  MoveL 1972 to (37.53, 7.97, 0.25) mm, rotated rx 180 ry 0 rz 90 deg; joints [74.413, -17.204, 82.136, 0, 25.068, 74.413]
  MoveL 1973 to (38.64, 6.94, -0.16) mm, rotated rx 180 ry 0 rz 90 deg; joints [74.39, -17.155, 82.02, 0, 25.135, 74.39]
  MoveL 1974 to (39.97, 6.21, -0.56) mm, rotated rx 180 ry 0 rz 90 deg; joints [74.379, -17.103, 81.894, 0, 25.209, 74.379]
  MoveL 1975 to (41.44, 5.79, -0.97) mm, rotated rx -180 ry 0 rz 90 deg; joints [74.379, -17.051, 81.765, 0, 25.286, 74.379]
  MoveL 1976 to (42.95, 5.71, -1.37) mm, rotated rx 180 ry 0 rz 90 deg; joints [74.389, -16.999, 81.638, 0, 25.361, 74.389]
  MoveL 1977 to (44.45, 5.96, -1.78) mm, rotated rx 180 ry 0 rz 90 deg; joints [74.411, -16.949, 81.519, 0, 25.43, 74.411]
  MoveL 1978 to (45.85, 6.54, -2.19) mm, rotated rx 180 ry 0 rz 90 deg; joints [74.441, -16.903, 81.414, 0, 25.489, 74.441]
  MoveL 1979 to (47.1, 7.42, -2.59) mm, rotated rx 180 ry 0 rz 90 deg; joints [74.48, -16.862, 81.327, 0, 25.535, 74.48]
  MoveL 1980 to (48.09, 8.56, -3) mm, rotated rx 180 ry 0 rz 90 deg; joints [74.525, -16.827, 81.263, 0, 25.564, 74.525]
  MoveL 1981 to (59.23, 24.09, -3) mm, rotated rx 180 ry 0 rz 90 deg; joints [75.111, -16.683, 80.75, 0, 25.933, 75.111]
  MoveL 1982 to (60.04, 25.3, -3) mm, rotated rx 180 ry 0 rz 90 deg; joints [75.156, -16.673, 80.714, 0, 25.959, 75.156]
  MoveC 1983 to (60.83, 30.5, -3) mm, rotated rx 180 ry 0 rz 90 deg; joints [75.327, -16.685, 80.757, 0, 25.928, 75.327] to (57.33, 34.43, -3) mm, rotated rx 180 ry 0 rz 90 deg; joints [75.423, -16.78, 81.093, 0, 25.686, 75.423]
  MoveC 1984 to (55.77, 34.77, -3) mm, rotated rx -180 ry 0 rz 90 deg; joints [75.421, -16.814, 81.216, 0, 25.598, 75.421] to (54.17, 34.86, -3) mm, rotated rx -180 ry 0 rz 90 deg; joints [75.41, -16.848, 81.336, 0, 25.512, 75.41]
  MoveL 1985 to (7.66, 33.6, -3) mm, rotated rx 180 ry 0 rz 90 deg; joints [74.974, -17.751, 84.687, 0, 23.065, 74.974]
  MoveC 1986 to (4.92, 33.05, -3) mm, rotated rx -180 ry 0 rz 90 deg; joints [74.933, -17.799, 84.871, 0, 22.928, 74.933] to (2.52, 31.63, -3) mm, rotated rx -180 ry 0 rz 90 deg; joints [74.865, -17.836, 85.014, 0, 22.822, 74.865]
  MoveC 1987 to (0.88, 28.58, -3) mm, rotated rx 180 ry 0 rz 90 deg; joints [74.751, -17.851, 85.072, 0, 22.779, 74.751] to (1.07, 25.11, -3) mm, rotated rx -180 ry 0 rz 90 deg; joints [74.64, -17.83, 84.991, 0, 22.839, 74.64]
  MoveL 1988 to (1.71, 23.22, -3) mm, rotated rx 180 ry 0 rz 90 deg; joints [74.584, -17.809, 84.909, 0, 22.9, 74.584]
  MoveL 1989 to (7.22, 8.05, -3) mm, rotated rx -180 ry 0 rz 90 deg; joints [74.142, -17.629, 84.216, 0, 23.413, 74.142]
  MoveL 1990 to (7.43, 7.5, -3) mm, rotated rx -180 ry 0 rz 90 deg; joints [74.126, -17.622, 84.189, 0, 23.432, 74.126]
  MoveC 1991 to (8.35, 5.81, -3) mm, rotated rx 180 ry 0 rz 90 deg; joints [74.08, -17.595, 84.09, 0, 23.506, 74.08] to (9.69, 4.43, -3) mm, rotated rx -180 ry 0 rz 90 deg; joints [74.048, -17.563, 83.966, 0, 23.597, 74.048]
  MoveL 1992 to (26.06, -8.32, -3) mm, rotated rx 180 ry 0 rz 90 deg; joints [73.791, -17.176, 82.524, 0, 24.652, 73.791]
  MoveL 1993 to (27.21, -9.18, -3) mm, rotated rx 180 ry 0 rz 90 deg; joints [73.774, -17.148, 82.422, 0, 24.726, 73.774]
  MoveC 1994 to (31.85, -10.43, -3) mm, rotated rx 180 ry 0 rz 90 deg; joints [73.778, -17.048, 82.058, 0, 24.99, 73.778] to (36.06, -8.1, -3) mm, rotated rx -180 ry 0 rz 90 deg; joints [73.89, -16.977, 81.801, 0, 25.176, 73.89]
  MoveL 1995 to (36.86, -7.11, -3) mm, rotated rx -180 ry 0 rz 90 deg; joints [73.929, -16.966, 81.763, 0, 25.204, 73.929]
  MoveL 1996 to (44.07, 2.95, -3) mm, rotated rx -180 ry 0 rz 90 deg; joints [74.312, -16.878, 81.444, 0, 25.434, 74.312]
  MoveL 1997 to (48.09, 8.56, -3) mm, rotated rx 180 ry 0 rz 90 deg; joints [74.525, -16.827, 81.263, 0, 25.564, 74.525]
  MoveL 1998 to (41.96, 12.96, -3) mm, rotated rx -180 ry 0 rz 90 deg; joints [74.611, -16.978, 81.804, 0, 25.174, 74.611]
  MoveL 1999 to (41.96, 12.96, 0) mm, rotated rx 180 ry 0 rz 90 deg; joints [74.611, -17.13, 81.905, 0, 25.225, 74.611]
  Establecer velocidad (1000.0 mm/s)
  MoveL 2000 to (41.96, 12.96, 10) mm, rotated rx 180 ry 0 rz 90 deg; joints [74.611, -17.635, 82.239, 0, 25.396, 74.611]
  Establecer velocidad (66.7 mm/s)
  MoveL 2001 to (27.12, 70.14, 10) mm, rotated rx -180 ry 0 rz 90 deg; joints [76.326, -18.224, 84.396, 0, 23.829, 76.326]
  MoveL 2002 to (27.12, 70.14, 0.25) mm, rotated rx -180 ry 0 rz 90 deg; joints [76.326, -17.727, 84.071, 0, 23.656, 76.326]
  MoveL 2003 to (27.33, 71.65, -0.16) mm, rotated rx 180 ry 0 rz 90 deg; joints [76.377, -17.71, 84.069, 0, 23.641, 76.377]
  MoveL 2004 to (27.16, 73.16, -0.56) mm, rotated rx -180 ry 0 rz 90 deg; joints [76.425, -17.699, 84.094, 0, 23.606, 76.425]
  MoveL 2005 to (26.67, 74.59, -0.97) mm, rotated rx 180 ry 0 rz 90 deg; joints [76.468, -17.694, 84.14, 0, 23.554, 76.468]
  MoveL 2006 to (25.87, 75.89, -1.37) mm, rotated rx 180 ry 0 rz 90 deg; joints [76.504, -17.695, 84.207, 0, 23.488, 76.504]
  MoveL 2007 to (24.81, 76.97, -1.78) mm, rotated rx -180 ry 0 rz 90 deg; joints [76.531, -17.699, 84.288, 0, 23.411, 76.531]
  MoveL 2008 to (23.53, 77.8, -2.19) mm, rotated rx 180 ry 0 rz 90 deg; joints [76.547, -17.706, 84.381, 0, 23.325, 76.547]
  MoveL 2009 to (22.1, 78.32, -2.59) mm, rotated rx 180 ry 0 rz 90 deg; joints [76.553, -17.715, 84.479, 0, 23.236, 76.553]
  MoveL 2010 to (20.6, 78.48, -3) mm, rotated rx -180 ry 0 rz 90 deg; joints [76.547, -17.723, 84.576, 0, 23.147, 76.547]
  MoveC 2011 to (-4.88, 78.78, -3) mm, rotated rx 180 ry 0 rz 90 deg; joints [76.355, -18.184, 86.391, 0, 21.793, 76.355] to (-30.36, 79, -3) mm, rotated rx -180 ry 0 rz 90 deg; joints [76.153, -18.615, 88.168, 0, 20.446, 76.153]
  MoveC 2012 to (-33.55, 78.8, -3) mm, rotated rx -180 ry 0 rz 90 deg; joints [76.12, -18.665, 88.385, 0, 20.281, 76.12] to (-36.69, 78.18, -3) mm, rotated rx 180 ry 0 rz 90 deg; joints [76.073, -18.713, 88.59, 0, 20.124, 76.073]
  MoveC 2013 to (-40.07, 74.26, -3) mm, rotated rx 180 ry 0 rz 90 deg; joints [75.912, -18.752, 88.754, 0, 19.997, 75.912] to (-39.33, 69.14, -3) mm, rotated rx 180 ry 0 rz 90 deg; joints [75.745, -18.719, 88.615, 0, 20.104, 75.745]
  MoveC 2014 to (-37.7, 67.63, -3) mm, rotated rx 180 ry 0 rz 90 deg; joints [75.709, -18.687, 88.477, 0, 20.21, 75.709] to (-35.91, 66.33, -3) mm, rotated rx 180 ry 0 rz 90 deg; joints [75.68, -18.653, 88.331, 0, 20.322, 75.68]
  MoveL 2015 to (-32.69, 64.28, -3) mm, rotated rx 180 ry 0 rz 90 deg; joints [75.639, -18.592, 88.074, 0, 20.518, 75.639]
  MoveL 2016 to (-16.58, 54.08, -3) mm, rotated rx 180 ry 0 rz 90 deg; joints [75.437, -18.279, 86.776, 0, 21.503, 75.437]
  MoveL 2017 to (-12.87, 51.72, -3) mm, rotated rx -180 ry 0 rz 90 deg; joints [75.391, -18.205, 86.473, 0, 21.731, 75.391]
  MoveC 2018 to (-9.92, 50.46, -3) mm, rotated rx 180 ry 0 rz 90 deg; joints [75.375, -18.148, 86.244, 0, 21.903, 75.375] to (-6.73, 50.2, -3) mm, rotated rx 180 ry 0 rz 90 deg; joints [75.393, -18.09, 86.015, 0, 22.075, 75.393]
  MoveC 2019 to (32.51, 53.09, -3) mm, rotated rx -180 ry 0 rz 90 deg; joints [75.816, -17.376, 83.265, 0, 24.111, 75.816] to (71.77, 55.83, -3) mm, rotated rx 180 ry 0 rz 90 deg; joints [76.217, -16.589, 80.419, 0, 26.17, 76.217]
  MoveC 2020 to (75.27, 57.49, -3) mm, rotated rx -180 ry 0 rz 90 deg; joints [76.296, -16.522, 80.186, 0, 26.336, 76.296] to (76.7, 61.09, -3) mm, rotated rx 180 ry 0 rz 90 deg; joints [76.421, -16.511, 80.145, 0, 26.366, 76.421]
  MoveL 2021 to (76.7, 71.55, -3) mm, rotated rx -180 ry 0 rz 90 deg; joints [76.753, -16.564, 80.332, 0, 26.232, 76.753]
  MoveL 2022 to (76.69, 72.49, -3) mm, rotated rx -180 ry 0 rz 90 deg; joints [76.783, -16.569, 80.35, 0, 26.219, 76.783]
  MoveC 2023 to (75.13, 76.06, -3) mm, rotated rx 180 ry 0 rz 90 deg; joints [76.884, -16.62, 80.53, 0, 26.091, 76.884] to (71.55, 77.57, -3) mm, rotated rx -180 ry 0 rz 90 deg; joints [76.906, -16.704, 80.825, 0, 25.879, 76.906]
  MoveC 2024 to (46.07, 78.07, -3) mm, rotated rx -180 ry 0 rz 90 deg; joints [76.73, -17.23, 82.722, 0, 24.508, 76.73] to (20.6, 78.48, -3) mm, rotated rx -180 ry 0 rz 90 deg; joints [76.547, -17.723, 84.576, 0, 23.147, 76.547]
  MoveL 2025 to (20.49, 70.93, -3) mm, rotated rx 180 ry 0 rz 90 deg; joints [76.299, -17.691, 84.453, 0, 23.238, 76.299]
  MoveL 2026 to (20.49, 70.93, 0) mm, rotated rx 180 ry 0 rz 90 deg; joints [76.299, -17.844, 84.554, 0, 23.29, 76.299]
  Establecer velocidad (1000.0 mm/s)
  MoveL 2027 to (20.49, 70.93, 10) mm, rotated rx -180 ry 0 rz 90 deg; joints [76.299, -18.355, 84.886, 0, 23.468, 76.299]
  Establecer velocidad (66.7 mm/s)
  MoveL 2028 to (27.11, 69.78, 10) mm, rotated rx -180 ry 0 rz 90 deg; joints [76.314, -18.223, 84.39, 0, 23.833, 76.314]
  MoveL 2029 to (27.11, 69.78, 0) mm, rotated rx 180 ry 0 rz 90 deg; joints [76.314, -17.713, 84.057, 0, 23.656, 76.314]
  MoveL 2030 to (27.32, 71.29, -0.41) mm, rotated rx -180 ry 0 rz 90 deg; joints [76.365, -17.696, 84.055, 0, 23.641, 76.365]
  MoveL 2031 to (27.16, 72.8, -0.81) mm, rotated rx -180 ry 0 rz 90 deg; joints [76.413, -17.685, 84.079, 0, 23.606, 76.413]
  MoveL 2032 to (26.67, 74.24, -1.22) mm, rotated rx 180 ry 0 rz 90 deg; joints [76.456, -17.68, 84.126, 0, 23.554, 76.456]
  MoveL 2033 to (25.87, 75.53, -1.63) mm, rotated rx -180 ry 0 rz 90 deg; joints [76.492, -17.68, 84.192, 0, 23.488, 76.492]
  MoveL 2034 to (24.81, 76.62, -2.03) mm, rotated rx 180 ry 0 rz 90 deg; joints [76.519, -17.685, 84.274, 0, 23.411, 76.519]
  MoveL 2035 to (23.53, 77.44, -2.44) mm, rotated rx -180 ry 0 rz 90 deg; joints [76.536, -17.692, 84.367, 0, 23.325, 76.536]
  MoveL 2036 to (22.1, 77.96, -2.84) mm, rotated rx -180 ry 0 rz 90 deg; joints [76.542, -17.7, 84.465, 0, 23.236, 76.542]
  MoveL 2037 to (20.59, 78.12, -3.25) mm, rotated rx 180 ry 0 rz 90 deg; joints [76.535, -17.708, 84.562, 0, 23.147, 76.535]
  MoveC 2038 to (-5.1, 78.43, -3.25) mm, rotated rx -180 ry 0 rz 90 deg; joints [76.341, -18.174, 86.392, 0, 21.782, 76.341] to (-30.8, 78.63, -3.25) mm, rotated rx 180 ry 0 rz 90 deg; joints [76.137, -18.607, 88.184, 0, 20.423, 76.137]
  MoveC 2039 to (-33.67, 78.43, -3.25) mm, rotated rx -180 ry 0 rz 90 deg; joints [76.107, -18.653, 88.378, 0, 20.275, 76.107] to (-36.48, 77.81, -3.25) mm, rotated rx 180 ry 0 rz 90 deg; joints [76.062, -18.695, 88.561, 0, 20.135, 76.062]
  MoveC 2040 to (-39.45, 73.96, -3.25) mm, rotated rx 180 ry 0 rz 90 deg; joints [75.907, -18.727, 88.698, 0, 20.029, 75.907] to (-38.79, 69.14, -3.25) mm, rotated rx 180 ry 0 rz 90 deg; joints [75.75, -18.698, 88.57, 0, 20.128, 75.75]
  MoveC 2041 to (-37.24, 67.74, -3.25) mm, rotated rx 180 ry 0 rz 90 deg; joints [75.716, -18.667, 88.439, 0, 20.228, 75.716] to (-35.54, 66.53, -3.25) mm, rotated rx -180 ry 0 rz 90 deg; joints [75.69, -18.635, 88.301, 0, 20.334, 75.69]
  MoveL 2042 to (-12.65, 52.03, -3.25) mm, rotated rx -180 ry 0 rz 90 deg; joints [75.403, -18.189, 86.455, 0, 21.734, 75.403]
  MoveC 2043 to (-9.84, 50.82, -3.25) mm, rotated rx 180 ry 0 rz 90 deg; joints [75.387, -18.135, 86.236, 0, 21.899, 75.387] to (-6.79, 50.56, -3.25) mm, rotated rx 180 ry 0 rz 90 deg; joints [75.405, -18.08, 86.018, 0, 22.062, 75.405]
  MoveC 2044 to (32.37, 53.44, -3.25) mm, rotated rx -180 ry 0 rz 90 deg; joints [75.827, -17.368, 83.274, 0, 24.094, 75.827] to (71.55, 56.18, -3.25) mm, rotated rx -180 ry 0 rz 90 deg; joints [76.226, -16.583, 80.434, 0, 26.149, 76.226]
  MoveC 2045 to (74.92, 57.7, -3.25) mm, rotated rx -180 ry 0 rz 90 deg; joints [76.3, -16.519, 80.208, 0, 26.31, 76.3] to (76.32, 61.12, -3.25) mm, rotated rx 180 ry 0 rz 90 deg; joints [76.419, -16.506, 80.165, 0, 26.341, 76.419]
  MoveL 2046 to (76.32, 71.55, -3.25) mm, rotated rx -180 ry 0 rz 90 deg; joints [76.75, -16.56, 80.352, 0, 26.207, 76.75]
  MoveL 2047 to (76.32, 72.32, -3.25) mm, rotated rx 180 ry 0 rz 90 deg; joints [76.774, -16.564, 80.366, 0, 26.197, 76.774]
  MoveC 2048 to (74.89, 75.73, -3.25) mm, rotated rx -180 ry 0 rz 90 deg; joints [76.872, -16.611, 80.534, 0, 26.077, 76.872] to (71.49, 77.19, -3.25) mm, rotated rx -180 ry 0 rz 90 deg; joints [76.893, -16.691, 80.814, 0, 25.876, 76.893]
  MoveC 2049 to (46.04, 77.71, -3.25) mm, rotated rx -180 ry 0 rz 90 deg; joints [76.718, -17.216, 82.709, 0, 24.507, 76.718] to (20.59, 78.12, -3.25) mm, rotated rx 180 ry 0 rz 90 deg; joints [76.535, -17.708, 84.562, 0, 23.147, 76.535]
  MoveL 2050 to (20.49, 70.57, -3.25) mm, rotated rx 180 ry 0 rz 90 deg; joints [76.287, -17.676, 84.438, 0, 23.238, 76.287]
  MoveL 2051 to (20.49, 70.57, -0.25) mm, rotated rx 180 ry 0 rz 90 deg; joints [76.287, -17.83, 84.539, 0, 23.29, 76.287]
  Establecer velocidad (1000.0 mm/s)
  MoveL 2052 to (20.49, 70.57, 10) mm, rotated rx -180 ry 0 rz 90 deg; joints [76.287, -18.353, 84.88, 0, 23.473, 76.287]
  Establecer velocidad (66.7 mm/s)
  MoveL 2053 to (38.92, 25.84, 10) mm, rotated rx -180 ry 0 rz 90 deg; joints [74.995, -17.768, 82.717, 0, 25.051, 74.995]
  MoveL 2054 to (38.92, 25.84, 0) mm, rotated rx -180 ry 0 rz 90 deg; joints [74.995, -17.262, 82.383, 0, 24.878, 74.995]
  MoveL 2055 to (39.07, 27.35, -0.41) mm, rotated rx 180 ry 0 rz 90 deg; joints [75.044, -17.246, 82.388, 0, 24.858, 75.044]
  MoveL 2056 to (38.84, 28.85, -0.81) mm, rotated rx 180 ry 0 rz 90 deg; joints [75.09, -17.238, 82.42, 0, 24.818, 75.09]
  MoveL 2057 to (38.29, 30.27, -1.22) mm, rotated rx 180 ry 0 rz 90 deg; joints [75.131, -17.236, 82.474, 0, 24.762, 75.131]
  MoveL 2058 to (37.44, 31.53, -1.63) mm, rotated rx 180 ry 0 rz 90 deg; joints [75.164, -17.239, 82.547, 0, 24.692, 75.164]
  MoveL 2059 to (36.33, 32.57, -2.03) mm, rotated rx 180 ry 0 rz 90 deg; joints [75.188, -17.246, 82.634, 0, 24.612, 75.188]
  MoveL 2060 to (35.02, 33.34, -2.44) mm, rotated rx -180 ry 0 rz 90 deg; joints [75.202, -17.255, 82.731, 0, 24.525, 75.202]
  MoveL 2061 to (33.58, 33.8, -2.84) mm, rotated rx 180 ry 0 rz 90 deg; joints [75.204, -17.266, 82.831, 0, 24.434, 75.204]
  MoveL 2062 to (32.06, 33.9, -3.25) mm, rotated rx 180 ry 0 rz 90 deg; joints [75.194, -17.275, 82.93, 0, 24.346, 75.194]
  MoveL 2063 to (7.73, 33.25, -3.25) mm, rotated rx 180 ry 0 rz 90 deg; joints [74.964, -17.736, 84.666, 0, 23.069, 74.964]
  MoveC 2064 to (5.09, 32.73, -3.25) mm, rotated rx 180 ry 0 rz 90 deg; joints [74.924, -17.782, 84.844, 0, 22.937, 74.924] to (2.77, 31.37, -3.25) mm, rotated rx 180 ry 0 rz 90 deg; joints [74.859, -17.817, 84.983, 0, 22.834, 74.859]
  MoveC 2065 to (1.25, 28.58, -3.25) mm, rotated rx -180 ry 0 rz 90 deg; joints [74.755, -17.831, 85.037, 0, 22.794, 74.755] to (1.36, 25.41, -3.25) mm, rotated rx -180 ry 0 rz 90 deg; joints [74.652, -17.813, 84.967, 0, 22.846, 74.652]
  MoveL 2066 to (1.75, 24.17, -3.25) mm, rotated rx -180 ry 0 rz 90 deg; joints [74.615, -17.8, 84.916, 0, 22.884, 74.615]
  MoveL 2067 to (7.7, 7.76, -3.25) mm, rotated rx 180 ry 0 rz 90 deg; joints [74.137, -17.605, 84.167, 0, 23.438, 74.137]
  MoveC 2068 to (8.6, 6.06, -3.25) mm, rotated rx -180 ry 0 rz 90 deg; joints [74.091, -17.579, 84.068, 0, 23.511, 74.091] to (9.94, 4.68, -3.25) mm, rotated rx 180 ry 0 rz 90 deg; joints [74.059, -17.546, 83.944, 0, 23.602, 74.059]
  MoveL 2069 to (27.37, -8.88, -3.25) mm, rotated rx -180 ry 0 rz 90 deg; joints [73.785, -17.134, 82.408, 0, 24.725, 73.785]
  MoveC 2070 to (31.35, -10.12, -3.25) mm, rotated rx 180 ry 0 rz 90 deg; joints [73.783, -17.047, 82.093, 0, 24.954, 73.783] to (35.17, -8.46, -3.25) mm, rotated rx -180 ry 0 rz 90 deg; joints [73.871, -16.98, 81.85, 0, 25.13, 73.871]
  MoveC 2071 to (36.01, -7.56, -3.25) mm, rotated rx 180 ry 0 rz 90 deg; joints [73.907, -16.968, 81.807, 0, 25.161, 73.907] to (36.77, -6.59, -3.25) mm, rotated rx -180 ry 0 rz 90 deg; joints [73.944, -16.959, 81.771, 0, 25.187, 73.944]
  MoveL 2072 to (58.85, 24.17, -3.25) mm, rotated rx 180 ry 0 rz 90 deg; joints [75.111, -16.679, 80.771, 0, 25.907, 75.111]
  MoveL 2073 to (59.23, 24.74, -3.25) mm, rotated rx 180 ry 0 rz 90 deg; joints [75.132, -16.674, 80.754, 0, 25.919, 75.132]
  MoveL 2074 to (59.48, 25.11, -3.25) mm, rotated rx 180 ry 0 rz 90 deg; joints [75.146, -16.671, 80.743, 0, 25.928, 75.146]
  MoveC 2075 to (60.29, 30.5, -3.25) mm, rotated rx -180 ry 0 rz 90 deg; joints [75.323, -16.683, 80.789, 0, 25.895, 75.323] to (56.39, 34.31, -3.25) mm, rotated rx 180 ry 0 rz 90 deg; joints [75.411, -16.786, 81.152, 0, 25.634, 75.411]
  MoveC 2076 to (54.97, 34.46, -3.25) mm, rotated rx -180 ry 0 rz 90 deg; joints [75.404, -16.816, 81.26, 0, 25.556, 75.404] to (53.54, 34.47, -3.25) mm, rotated rx -180 ry 0 rz 90 deg; joints [75.393, -16.846, 81.366, 0, 25.48, 75.393]
  MoveL 2077 to (32.06, 33.9, -3.25) mm, rotated rx 180 ry 0 rz 90 deg; joints [75.194, -17.275, 82.93, 0, 24.346, 75.194]
  MoveL 2078 to (32.27, 26.35, -3.25) mm, rotated rx 180 ry 0 rz 90 deg; joints [74.954, -17.232, 82.769, 0, 24.463, 74.954]
  MoveL 2079 to (32.27, 26.35, -0.25) mm, rotated rx -180 ry 0 rz 90 deg; joints [74.954, -17.384, 82.87, 0, 24.515, 74.954]
  Establecer velocidad (1000.0 mm/s)
  MoveL 2080 to (32.27, 26.35, 10) mm, rotated rx -180 ry 0 rz 90 deg; joints [74.954, -17.904, 83.211, 0, 24.693, 74.954]
  Establecer velocidad (66.7 mm/s)
  MoveL 2081 to (68.53, -31.53, 10) mm, rotated rx 180 ry 0 rz 90 deg; joints [73.455, -16.795, 79.319, 0, 27.477, 73.455]
  MoveL 2082 to (68.53, -31.53, 0) mm, rotated rx 180 ry 0 rz 90 deg; joints [73.455, -16.295, 78.983, 0, 27.312, 73.455]
  MoveL 2083 to (70.03, -31.71, -0.41) mm, rotated rx -180 ry 0 rz 90 deg; joints [73.463, -16.24, 78.852, 0, 27.388, 73.463]
  MoveL 2084 to (71.54, -31.53, -0.81) mm, rotated rx -180 ry 0 rz 90 deg; joints [73.482, -16.187, 78.728, 0, 27.459, 73.482]
  MoveL 2085 to (72.97, -31.02, -1.22) mm, rotated rx 180 ry 0 rz 90 deg; joints [73.511, -16.138, 78.617, 0, 27.521, 73.511]
  MoveL 2086 to (74.25, -30.21, -1.63) mm, rotated rx 180 ry 0 rz 90 deg; joints [73.548, -16.095, 78.525, 0, 27.57, 73.548]
  MoveL 2087 to (75.33, -29.13, -2.03) mm, rotated rx -180 ry 0 rz 90 deg; joints [73.591, -16.058, 78.454, 0, 27.604, 73.591]
  MoveL 2088 to (76.13, -27.84, -2.44) mm, rotated rx 180 ry 0 rz 90 deg; joints [73.638, -16.028, 78.408, 0, 27.62, 73.638]
  MoveL 2089 to (76.63, -26.4, -2.84) mm, rotated rx -180 ry 0 rz 90 deg; joints [73.687, -16.006, 78.388, 0, 27.618, 73.687]
  MoveL 2090 to (76.77, -24.89, -3.25) mm, rotated rx -180 ry 0 rz 90 deg; joints [73.735, -15.992, 78.397, 0, 27.595, 73.735]
  MoveL 2091 to (76.77, -5.21, -3.25) mm, rotated rx 180 ry 0 rz 90 deg; joints [74.344, -16.118, 78.824, 0, 27.294, 74.344]
  MoveL 2092 to (76.75, -3.81, -3.25) mm, rotated rx -180 ry 0 rz 90 deg; joints [74.387, -16.127, 78.855, 0, 27.272, 74.387]
  MoveC 2093 to (76.11, -1.37, -3.25) mm, rotated rx -180 ry 0 rz 90 deg; joints [74.457, -16.156, 78.955, 0, 27.201, 74.457] to (74.39, 0.48, -3.25) mm, rotated rx 180 ry 0 rz 90 deg; joints [74.5, -16.205, 79.124, 0, 27.082, 74.5]
  MoveC 2094 to (71.22, 1.94, -3.25) mm, rotated rx -180 ry 0 rz 90 deg; joints [74.518, -16.284, 79.394, 0, 26.89, 74.518] to (67.76, 1.45, -3.25) mm, rotated rx 180 ry 0 rz 90 deg; joints [74.473, -16.356, 79.644, 0, 26.712, 74.473]
  MoveL 2095 to (67.48, 1.21, -3.25) mm, rotated rx 180 ry 0 rz 90 deg; joints [74.463, -16.361, 79.66, 0, 26.701, 74.463]
  MoveL 2096 to (65.86, -0.82, -3.25) mm, rotated rx 180 ry 0 rz 90 deg; joints [74.385, -16.384, 79.739, 0, 26.645, 74.385]
  MoveL 2097 to (63.34, -4.26, -3.25) mm, rotated rx -180 ry 0 rz 90 deg; joints [74.256, -16.417, 79.855, 0, 26.562, 74.256]
  MoveL 2098 to (51.65, -20.31, -3.25) mm, rotated rx 180 ry 0 rz 90 deg; joints [73.648, -16.568, 80.383, 0, 26.186, 73.648]
  MoveL 2099 to (49.96, -22.62, -3.25) mm, rotated rx -180 ry 0 rz 90 deg; joints [73.561, -16.59, 80.457, 0, 26.132, 73.561]
  MoveC 2100 to (48.85, -26.25, -3.25) mm, rotated rx 180 ry 0 rz 90 deg; joints [73.437, -16.59, 80.46, 0, 26.13, 73.437] to (50.23, -29.78, -3.25) mm, rotated rx -180 ry 0 rz 90 deg; joints [73.34, -16.539, 80.279, 0, 26.259, 73.34]
  MoveL 2101 to (50.7, -30.33, -3.25) mm, rotated rx -180 ry 0 rz 90 deg; joints [73.327, -16.526, 80.233, 0, 26.293, 73.327]
  MoveL 2102 to (66.21, -47.86, -3.25) mm, rotated rx 180 ry 0 rz 90 deg; joints [72.929, -16.074, 78.676, 0, 27.398, 72.929]
  MoveL 2103 to (67.31, -49.04, -3.25) mm, rotated rx 180 ry 0 rz 90 deg; joints [72.903, -16.042, 78.566, 0, 27.476, 72.903]
  MoveC 2104 to (68.75, -50.03, -3.25) mm, rotated rx 180 ry 0 rz 90 deg; joints [72.887, -16.003, 78.433, 0, 27.569, 72.887] to (70.48, -50.31, -3.25) mm, rotated rx 180 ry 0 rz 90 deg; joints [72.894, -15.962, 78.296, 0, 27.666, 72.894]
  MoveC 2105 to (74.16, -49.02, -3.25) mm, rotated rx -180 ry 0 rz 90 deg; joints [72.968, -15.888, 78.048, 0, 27.841, 72.968] to (76.56, -45.96, -3.25) mm, rotated rx -180 ry 0 rz 90 deg; joints [73.085, -15.855, 77.936, 0, 27.919, 73.085]
  MoveL 2106 to (76.65, -45.49, -3.25) mm, rotated rx 180 ry 0 rz 90 deg; joints [73.1, -15.856, 77.94, 0, 27.917, 73.1]
  MoveL 2107 to (76.77, -43.12, -3.25) mm, rotated rx 180 ry 0 rz 90 deg; joints [73.174, -15.87, 77.986, 0, 27.884, 73.174]
  MoveL 2108 to (76.77, -24.89, -3.25) mm, rotated rx -180 ry 0 rz 90 deg; joints [73.735, -15.992, 78.397, 0, 27.595, 73.735]
  MoveL 2109 to (69.22, -24.89, -3.25) mm, rotated rx -180 ry 0 rz 90 deg; joints [73.666, -16.16, 78.968, 0, 27.192, 73.666]
  MoveL 2110 to (69.22, -24.89, -0.25) mm, rotated rx 180 ry 0 rz 90 deg; joints [73.666, -16.31, 79.07, 0, 27.24, 73.666]
  Establecer velocidad (1000.0 mm/s)
  MoveL 2111 to (69.22, -24.89, 10) mm, rotated rx -180 ry 0 rz 90 deg; joints [73.666, -16.824, 79.414, 0, 27.409, 73.666]
  Establecer velocidad (66.7 mm/s)
  MoveL 2112 to (18.39, -70.07, 10) mm, rotated rx 180 ry 0 rz 90 deg; joints [71.768, -17.604, 82.128, 0, 25.476, 71.768]
  MoveL 2113 to (18.39, -70.07, 0) mm, rotated rx 180 ry 0 rz 90 deg; joints [71.768, -17.099, 81.794, 0, 25.305, 71.768]
  MoveL 2114 to (18.22, -71.58, -0.41) mm, rotated rx 180 ry 0 rz 90 deg; joints [71.719, -17.072, 81.757, 0, 25.315, 71.719]
  MoveL 2115 to (18.42, -73.08, -0.81) mm, rotated rx 180 ry 0 rz 90 deg; joints [71.674, -17.037, 81.693, 0, 25.344, 71.674]
  MoveL 2116 to (18.94, -74.51, -1.22) mm, rotated rx 180 ry 0 rz 90 deg; joints [71.635, -16.996, 81.607, 0, 25.39, 71.635]
  MoveL 2117 to (19.77, -75.78, -1.63) mm, rotated rx 180 ry 0 rz 90 deg; joints [71.604, -16.951, 81.502, 0, 25.448, 71.604]
  MoveL 2118 to (20.86, -76.84, -2.03) mm, rotated rx 180 ry 0 rz 90 deg; joints [71.582, -16.901, 81.384, 0, 25.517, 71.582]
  MoveL 2119 to (22.16, -77.63, -2.44) mm, rotated rx 180 ry 0 rz 90 deg; joints [71.571, -16.849, 81.257, 0, 25.592, 71.571]
  MoveL 2120 to (23.6, -78.12, -2.84) mm, rotated rx -180 ry 0 rz 90 deg; joints [71.571, -16.795, 81.127, 0, 25.669, 71.571]
  MoveL 2121 to (25.11, -78.24, -3.25) mm, rotated rx -180 ry 0 rz 90 deg; joints [71.583, -16.743, 81, 0, 25.743, 71.583]
  MoveL 2122 to (46.91, -78.02, -3.25) mm, rotated rx 180 ry 0 rz 90 deg; joints [71.812, -16.286, 79.402, 0, 26.884, 71.812]
  MoveL 2123 to (53.54, -77.93, -3.25) mm, rotated rx 180 ry 0 rz 90 deg; joints [71.882, -16.143, 78.91, 0, 27.233, 71.882]
  MoveC 2124 to (54.99, -77.82, -3.25) mm, rotated rx 180 ry 0 rz 90 deg; joints [71.9, -16.112, 78.805, 0, 27.307, 71.9] to (56.39, -77.45, -3.25) mm, rotated rx -180 ry 0 rz 90 deg; joints [71.925, -16.084, 78.71, 0, 27.374, 71.925]
  MoveC 2125 to (59.33, -74.05, -3.25) mm, rotated rx -180 ry 0 rz 90 deg; joints [72.059, -16.044, 78.572, 0, 27.472, 72.059] to (59.23, -69.56, -3.25) mm, rotated rx -180 ry 0 rz 90 deg; joints [72.195, -16.078, 78.688, 0, 27.39, 72.195]
  MoveL 2126 to (58.7, -68.7, -3.25) mm, rotated rx 180 ry 0 rz 90 deg; joints [72.216, -16.095, 78.748, 0, 27.347, 72.216]
  MoveL 2127 to (58.28, -68.13, -3.25) mm, rotated rx -180 ry 0 rz 90 deg; joints [72.23, -16.109, 78.793, 0, 27.315, 72.23]
  MoveL 2128 to (57.99, -67.76, -3.25) mm, rotated rx 180 ry 0 rz 90 deg; joints [72.238, -16.118, 78.824, 0, 27.294, 72.238]
  MoveL 2129 to (57.33, -66.96, -3.25) mm, rotated rx -180 ry 0 rz 90 deg; joints [72.256, -16.138, 78.892, 0, 27.245, 72.256]
  MoveL 2130 to (28.71, -33.86, -3.25) mm, rotated rx -180 ry 0 rz 90 deg; joints [73.007, -16.958, 81.769, 0, 25.189, 73.007]
  MoveL 2131 to (28.24, -33.34, -3.25) mm, rotated rx 180 ry 0 rz 90 deg; joints [73.019, -16.971, 81.815, 0, 25.156, 73.019]
  MoveL 2132 to (26.25, -31.75, -3.25) mm, rotated rx 180 ry 0 rz 90 deg; joints [73.05, -17.02, 81.995, 0, 25.025, 73.05]
  MoveL 2133 to (14.39, -22.27, -3.25) mm, rotated rx 180 ry 0 rz 90 deg; joints [73.237, -17.31, 83.059, 0, 24.251, 73.237]
  MoveL 2134 to (13.74, -21.74, -3.25) mm, rotated rx -180 ry 0 rz 90 deg; joints [73.248, -17.326, 83.117, 0, 24.209, 73.248]
  MoveC 2135 to (11.95, -20.53, -3.25) mm, rotated rx 180 ry 0 rz 90 deg; joints [73.269, -17.368, 83.272, 0, 24.096, 73.269] to (9.95, -19.72, -3.25) mm, rotated rx 180 ry 0 rz 90 deg; joints [73.276, -17.411, 83.433, 0, 23.978, 73.276]
  MoveC 2136 to (6.07, -20.02, -3.25) mm, rotated rx -180 ry 0 rz 90 deg; joints [73.229, -17.483, 83.703, 0, 23.779, 73.229] to (3.32, -22.77, -3.25) mm, rotated rx -180 ry 0 rz 90 deg; joints [73.114, -17.519, 83.84, 0, 23.679, 73.114]
  MoveC 2137 to (2.76, -24.15, -3.25) mm, rotated rx 180 ry 0 rz 90 deg; joints [73.064, -17.522, 83.85, 0, 23.672, 73.064] to (2.32, -25.57, -3.25) mm, rotated rx -180 ry 0 rz 90 deg; joints [73.015, -17.522, 83.851, 0, 23.671, 73.015]
  MoveL 2138 to (-9.62, -70.6, -3.25) mm, rotated rx -180 ry 0 rz 90 deg; joints [71.458, -17.475, 83.674, 0, 23.801, 71.458]
  MoveC 2139 to (-9.66, -73.59, -3.25) mm, rotated rx -180 ry 0 rz 90 deg; joints [71.363, -17.457, 83.606, 0, 23.851, 71.363] to (-8.34, -76.29, -3.25) mm, rotated rx -180 ry 0 rz 90 deg; joints [71.292, -17.415, 83.448, 0, 23.966, 71.292]
  MoveC 2140 to (-6.05, -77.88, -3.25) mm, rotated rx -180 ry 0 rz 90 deg; joints [71.266, -17.361, 83.247, 0, 24.114, 71.266] to (-3.32, -78.49, -3.25) mm, rotated rx 180 ry 0 rz 90 deg; joints [71.276, -17.305, 83.039, 0, 24.266, 71.276]
  MoveL 2141 to (-2.37, -78.52, -3.25) mm, rotated rx 180 ry 0 rz 90 deg; joints [71.285, -17.287, 82.971, 0, 24.316, 71.285]
  MoveL 2142 to (25.11, -78.24, -3.25) mm, rotated rx -180 ry 0 rz 90 deg; joints [71.583, -16.743, 81, 0, 25.743, 71.583]
  MoveL 2143 to (25.04, -70.69, -3.25) mm, rotated rx 180 ry 0 rz 90 deg; joints [71.817, -16.796, 81.187, 0, 25.608, 71.817]
  MoveL 2144 to (25.04, -70.69, -0.25) mm, rotated rx 180 ry 0 rz 90 deg; joints [71.817, -16.947, 81.289, 0, 25.659, 71.817]
  Establecer velocidad (1000.0 mm/s)
  MoveL 2145 to (25.04, -70.69, 10) mm, rotated rx -180 ry 0 rz 90 deg; joints [71.817, -17.464, 81.631, 0, 25.833, 71.817]
  Establecer velocidad (66.7 mm/s)
  MoveL 2146 to (-70.97, -45.14, 10) mm, rotated rx 180 ry 0 rz 90 deg; joints [71.619, -19.366, 88.925, 0, 20.441, 71.619]
  MoveL 2147 to (-70.97, -45.14, 0) mm, rotated rx -180 ry 0 rz 90 deg; joints [71.619, -18.847, 88.593, 0, 20.254, 71.619]
  MoveL 2148 to (-72.48, -44.95, -0.41) mm, rotated rx 180 ry 0 rz 90 deg; joints [71.609, -18.85, 88.684, 0, 20.166, 71.609]
  MoveL 2149 to (-73.99, -45.13, -0.81) mm, rotated rx 180 ry 0 rz 90 deg; joints [71.586, -18.851, 88.768, 0, 20.084, 71.586]
  MoveL 2150 to (-75.42, -45.65, -1.22) mm, rotated rx 180 ry 0 rz 90 deg; joints [71.554, -18.85, 88.838, 0, 20.012, 71.554]
  MoveL 2151 to (-76.7, -46.46, -1.63) mm, rotated rx 180 ry 0 rz 90 deg; joints [71.513, -18.844, 88.892, 0, 19.952, 71.513]
  MoveL 2152 to (-77.77, -47.54, -2.03) mm, rotated rx -180 ry 0 rz 90 deg; joints [71.465, -18.834, 88.926, 0, 19.908, 71.465]
  MoveL 2153 to (-78.57, -48.83, -2.44) mm, rotated rx -180 ry 0 rz 90 deg; joints [71.413, -18.819, 88.937, 0, 19.882, 71.413]
  MoveL 2154 to (-79.07, -50.27, -2.84) mm, rotated rx -180 ry 0 rz 90 deg; joints [71.36, -18.798, 88.925, 0, 19.873, 71.36]
  MoveL 2155 to (-79.21, -51.78, -3.25) mm, rotated rx -180 ry 0 rz 90 deg; joints [71.309, -18.771, 88.886, 0, 19.885, 71.309]
  MoveL 2156 to (-79.21, -70.6, -3.25) mm, rotated rx -180 ry 0 rz 90 deg; joints [70.689, -18.67, 88.453, 0, 20.217, 70.689]
  MoveL 2157 to (-79.17, -71.49, -3.25) mm, rotated rx 180 ry 0 rz 90 deg; joints [70.66, -18.665, 88.43, 0, 20.235, 70.66]
  MoveC 2158 to (-77.88, -75.33, -3.25) mm, rotated rx 180 ry 0 rz 90 deg; joints [70.549, -18.623, 88.253, 0, 20.37, 70.549] to (-74.72, -77.87, -3.25) mm, rotated rx -180 ry 0 rz 90 deg; joints [70.503, -18.559, 87.982, 0, 20.578, 70.503]
  MoveC 2159 to (-72.91, -78.42, -3.25) mm, rotated rx -180 ry 0 rz 90 deg; joints [70.506, -18.527, 87.847, 0, 20.68, 70.506] to (-71.03, -78.6, -3.25) mm, rotated rx 180 ry 0 rz 90 deg; joints [70.522, -18.496, 87.716, 0, 20.78, 70.522]
  MoveL 2160 to (-42.17, -78.36, -3.25) mm, rotated rx 180 ry 0 rz 90 deg; joints [70.856, -18.015, 85.759, 0, 22.256, 70.856]
  MoveL 2161 to (-35.3, -78.3, -3.25) mm, rotated rx 180 ry 0 rz 90 deg; joints [70.935, -17.895, 85.286, 0, 22.609, 70.935]
  MoveC 2162 to (-30.58, -76.65, -3.25) mm, rotated rx 180 ry 0 rz 90 deg; joints [71.039, -17.821, 84.999, 0, 22.823, 71.039] to (-27.84, -72.47, -3.25) mm, rotated rx -180 ry 0 rz 90 deg; joints [71.203, -17.798, 84.907, 0, 22.891, 71.203]
  MoveL 2163 to (-15.17, -23.85, -3.25) mm, rotated rx -180 ry 0 rz 90 deg; joints [72.898, -17.853, 85.123, 0, 22.731, 72.898]
  MoveC 2164 to (-14.92, -20.63, -3.25) mm, rotated rx -180 ry 0 rz 90 deg; joints [73.004, -17.866, 85.174, 0, 22.692, 73.004] to (-15.82, -17.53, -3.25) mm, rotated rx -180 ry 0 rz 90 deg; joints [73.096, -17.899, 85.303, 0, 22.596, 73.096]
  MoveC 2165 to (-19, -14.74, -3.25) mm, rotated rx -180 ry 0 rz 90 deg; joints [73.155, -17.971, 85.585, 0, 22.386, 73.155] to (-23.22, -14.28, -3.25) mm, rotated rx -180 ry 0 rz 90 deg; joints [73.128, -18.048, 85.889, 0, 22.159, 73.128]
  MoveL 2166 to (-24.17, -14.45, -3.25) mm, rotated rx 180 ry 0 rz 90 deg; joints [73.113, -18.064, 85.951, 0, 22.112, 73.113]
  MoveL 2167 to (-72.49, -24.72, -3.25) mm, rotated rx -180 ry 0 rz 90 deg; joints [72.279, -18.804, 89.032, 0, 19.772, 72.279]
  MoveL 2168 to (-73.38, -24.94, -3.25) mm, rotated rx -180 ry 0 rz 90 deg; joints [72.263, -18.817, 89.086, 0, 19.73, 72.263]
  MoveC 2169 to (-77.48, -27.52, -3.25) mm, rotated rx 180 ry 0 rz 90 deg; joints [72.133, -18.867, 89.305, 0, 19.562, 72.133] to (-79.19, -32.06, -3.25) mm, rotated rx -180 ry 0 rz 90 deg; joints [71.963, -18.87, 89.321, 0, 19.549, 71.963]
  MoveL 2170 to (-79.21, -32.69, -3.25) mm, rotated rx 180 ry 0 rz 90 deg; joints [71.942, -18.868, 89.309, 0, 19.559, 71.942]
  MoveL 2171 to (-79.21, -51.78, -3.25) mm, rotated rx -180 ry 0 rz 90 deg; joints [71.309, -18.771, 88.886, 0, 19.885, 71.309]
  MoveL 2172 to (-71.66, -51.78, -3.25) mm, rotated rx 180 ry 0 rz 90 deg; joints [71.393, -18.653, 88.381, 0, 20.273, 71.393]
  MoveL 2173 to (-71.66, -51.78, -0.25) mm, rotated rx 180 ry 0 rz 90 deg; joints [71.393, -18.809, 88.482, 0, 20.328, 71.393]
  Establecer velocidad (1000.0 mm/s)
  MoveL 2174 to (-71.66, -51.78, 10) mm, rotated rx 180 ry 0 rz 90 deg; joints [71.393, -19.342, 88.822, 0, 20.52, 71.393]
  Establecer velocidad (66.7 mm/s)
  MoveL 2175 to (-70.97, 36.02, 10) mm, rotated rx 180 ry 0 rz 90 deg; joints [74.338, -19.751, 90.592, 0, 19.159, 74.338]
  MoveL 2176 to (-70.97, 36.02, 0) mm, rotated rx -180 ry 0 rz 90 deg; joints [74.338, -19.227, 90.259, 0, 18.967, 74.338]
  MoveL 2177 to (-72.48, 36.2, -0.41) mm, rotated rx 180 ry 0 rz 90 deg; joints [74.33, -19.228, 90.35, 0, 18.878, 74.33]
  MoveL 2178 to (-73.99, 36.02, -0.81) mm, rotated rx 180 ry 0 rz 90 deg; joints [74.309, -19.229, 90.434, 0, 18.795, 74.309]
  MoveL 2179 to (-75.42, 35.51, -1.22) mm, rotated rx 180 ry 0 rz 90 deg; joints [74.278, -19.226, 90.506, 0, 18.72, 74.278]
  MoveL 2180 to (-76.7, 34.69, -1.63) mm, rotated rx 180 ry 0 rz 90 deg; joints [74.238, -19.22, 90.562, 0, 18.658, 74.238]
  MoveL 2181 to (-77.77, 33.61, -2.03) mm, rotated rx -180 ry 0 rz 90 deg; joints [74.191, -19.21, 90.6, 0, 18.61, 74.191]
  MoveL 2182 to (-78.57, 32.32, -2.44) mm, rotated rx -180 ry 0 rz 90 deg; joints [74.139, -19.195, 90.615, 0, 18.58, 74.139]
  MoveL 2183 to (-79.07, 30.89, -2.84) mm, rotated rx 180 ry 0 rz 90 deg; joints [74.085, -19.175, 90.607, 0, 18.567, 74.085]
  MoveL 2184 to (-79.21, 29.38, -3.25) mm, rotated rx -180 ry 0 rz 90 deg; joints [74.032, -19.149, 90.574, 0, 18.575, 74.032]
  MoveL 2185 to (-79.21, 0.47, -3.25) mm, rotated rx -180 ry 0 rz 90 deg; joints [73.053, -19.024, 90.006, 0, 19.018, 73.053]
  MoveC 2186 to (-77.93, -3.81, -3.25) mm, rotated rx -180 ry 0 rz 90 deg; joints [72.922, -18.986, 89.833, 0, 19.153, 72.922] to (-74.39, -6.55, -3.25) mm, rotated rx -180 ry 0 rz 90 deg; joints [72.867, -18.92, 89.541, 0, 19.379, 72.867]
  MoveC 2187 to (-72.04, -6.99, -3.25) mm, rotated rx 180 ry 0 rz 90 deg; joints [72.876, -18.882, 89.374, 0, 19.508, 72.876] to (-69.65, -6.81, -3.25) mm, rotated rx -180 ry 0 rz 90 deg; joints [72.907, -18.847, 89.218, 0, 19.629, 72.907]
  MoveL 2188 to (-26.06, 3.21, -3.25) mm, rotated rx 180 ry 0 rz 90 deg; joints [73.672, -18.188, 86.449, 0, 21.739, 73.672]
  MoveL 2189 to (-19.68, 4.69, -3.25) mm, rotated rx 180 ry 0 rz 90 deg; joints [73.782, -18.085, 86.035, 0, 22.049, 73.782]
  MoveC 2190 to (-14.99, 8.13, -3.25) mm, rotated rx 180 ry 0 rz 90 deg; joints [73.939, -18.02, 85.777, 0, 22.243, 73.939] to (-14.25, 13.91, -3.25) mm, rotated rx -180 ry 0 rz 90 deg; joints [74.134, -18.036, 85.841, 0, 22.195, 74.134]
  MoveL 2191 to (-14.47, 14.69, -3.25) mm, rotated rx 180 ry 0 rz 90 deg; joints [74.158, -18.044, 85.872, 0, 22.172, 74.158]
  MoveL 2192 to (-18.48, 25.9, -3.25) mm, rotated rx 180 ry 0 rz 90 deg; joints [74.489, -18.169, 86.372, 0, 21.797, 74.489]
  MoveL 2193 to (-21.25, 33.66, -3.25) mm, rotated rx -180 ry 0 rz 90 deg; joints [74.72, -18.253, 86.714, 0, 21.539, 74.72]
  MoveC 2194 to (-22.55, 35.98, -3.25) mm, rotated rx 180 ry 0 rz 90 deg; joints [74.785, -18.286, 86.847, 0, 21.439, 74.785] to (-24.52, 37.76, -3.25) mm, rotated rx 180 ry 0 rz 90 deg; joints [74.826, -18.328, 87.018, 0, 21.31, 74.826]
  MoveL 2195 to (-65.86, 64.28, -3.25) mm, rotated rx 180 ry 0 rz 90 deg; joints [75.348, -19.094, 90.321, 0, 18.773, 75.348]
  MoveL 2196 to (-66.81, 64.87, -3.25) mm, rotated rx 180 ry 0 rz 90 deg; joints [75.36, -19.11, 90.395, 0, 18.715, 75.36]
  MoveC 2197 to (-69.08, 66, -3.25) mm, rotated rx 180 ry 0 rz 90 deg; joints [75.378, -19.148, 90.567, 0, 18.581, 75.378] to (-71.55, 66.59, -3.25) mm, rotated rx 180 ry 0 rz 90 deg; joints [75.376, -19.186, 90.742, 0, 18.444, 75.376]
  MoveC 2198 to (-75.93, 65.62, -3.25) mm, rotated rx 180 ry 0 rz 90 deg; joints [75.304, -19.245, 91.018, 0, 18.227, 75.304] to (-78.69, 62.07, -3.25) mm, rotated rx 180 ry 0 rz 90 deg; joints [75.156, -19.271, 91.139, 0, 18.132, 75.156]
  MoveC 2199 to (-79.1, 60.2, -3.25) mm, rotated rx -180 ry 0 rz 90 deg; joints [75.088, -19.27, 91.133, 0, 18.136, 75.088] to (-79.21, 58.28, -3.25) mm, rotated rx 180 ry 0 rz 90 deg; joints [75.021, -19.264, 91.107, 0, 18.157, 75.021]
  MoveL 2200 to (-79.21, 29.38, -3.25) mm, rotated rx -180 ry 0 rz 90 deg; joints [74.032, -19.149, 90.574, 0, 18.575, 74.032]
  MoveL 2201 to (-71.66, 29.38, -3.25) mm, rotated rx 180 ry 0 rz 90 deg; joints [74.106, -19.039, 90.07, 0, 18.968, 74.106]
  MoveL 2202 to (-71.66, 29.38, -0.25) mm, rotated rx 180 ry 0 rz 90 deg; joints [74.106, -19.196, 90.171, 0, 19.024, 74.106]
  Establecer velocidad (1000.0 mm/s)
  MoveL 2203 to (-71.66, 29.38, 10) mm, rotated rx -180 ry 0 rz 90 deg; joints [74.106, -19.733, 90.513, 0, 19.22, 74.106]
  Establecer velocidad (66.7 mm/s)
  MoveL 2204 to (-70.64, 36.02, 10) mm, rotated rx 180 ry 0 rz 90 deg; joints [74.341, -19.746, 90.57, 0, 19.176, 74.341]
  MoveL 2205 to (-70.64, 36.02, -0.25) mm, rotated rx 180 ry 0 rz 90 deg; joints [74.341, -19.209, 90.229, 0, 18.98, 74.341]
  MoveL 2206 to (-72.14, 36.2, -0.66) mm, rotated rx 180 ry 0 rz 90 deg; joints [74.333, -19.21, 90.319, 0, 18.891, 74.333]
  MoveL 2207 to (-73.65, 36.02, -1.06) mm, rotated rx -180 ry 0 rz 90 deg; joints [74.312, -19.211, 90.403, 0, 18.808, 74.312]
  MoveL 2208 to (-75.08, 35.51, -1.47) mm, rotated rx -180 ry 0 rz 90 deg; joints [74.281, -19.208, 90.475, 0, 18.733, 74.281]
  MoveL 2209 to (-76.36, 34.69, -1.87) mm, rotated rx -180 ry 0 rz 90 deg; joints [74.241, -19.202, 90.532, 0, 18.67, 74.241]
  MoveL 2210 to (-77.43, 33.61, -2.28) mm, rotated rx 180 ry 0 rz 90 deg; joints [74.194, -19.192, 90.569, 0, 18.623, 74.194]
  MoveL 2211 to (-78.24, 32.32, -2.69) mm, rotated rx -180 ry 0 rz 90 deg; joints [74.142, -19.177, 90.585, 0, 18.592, 74.142]
  MoveL 2212 to (-78.74, 30.89, -3.09) mm, rotated rx 180 ry 0 rz 90 deg; joints [74.088, -19.157, 90.577, 0, 18.58, 74.088]
  MoveL 2213 to (-78.87, 29.38, -3.5) mm, rotated rx 180 ry 0 rz 90 deg; joints [74.036, -19.131, 90.544, 0, 18.588, 74.036]
  MoveL 2214 to (-78.87, 0.33, -3.5) mm, rotated rx -180 ry 0 rz 90 deg; joints [73.052, -19.006, 89.972, 0, 19.034, 73.052]
  MoveC 2215 to (-77.22, -4.17, -3.5) mm, rotated rx -180 ry 0 rz 90 deg; joints [72.917, -18.961, 89.77, 0, 19.19, 72.917] to (-73.06, -6.55, -3.5) mm, rotated rx -180 ry 0 rz 90 deg; joints [72.881, -18.887, 89.443, 0, 19.444, 72.881]
  MoveC 2216 to (-71.35, -6.67, -3.5) mm, rotated rx 180 ry 0 rz 90 deg; joints [72.894, -18.861, 89.326, 0, 19.534, 72.894] to (-69.65, -6.46, -3.5) mm, rotated rx -180 ry 0 rz 90 deg; joints [72.918, -18.836, 89.217, 0, 19.619, 72.918]
  MoveL 2217 to (-68.7, -6.25, -3.5) mm, rotated rx 180 ry 0 rz 90 deg; joints [72.935, -18.822, 89.157, 0, 19.665, 72.935]
  MoveL 2218 to (-19.72, 5.05, -3.5) mm, rotated rx 180 ry 0 rz 90 deg; joints [73.793, -18.074, 86.037, 0, 22.038, 73.793]
  MoveC 2219 to (-15.28, 8.29, -3.5) mm, rotated rx 180 ry 0 rz 90 deg; joints [73.941, -18.013, 85.792, 0, 22.221, 73.941] to (-14.57, 13.74, -3.5) mm, rotated rx 180 ry 0 rz 90 deg; joints [74.126, -18.028, 85.851, 0, 22.176, 74.126]
  MoveL 2220 to (-14.83, 14.69, -3.5) mm, rotated rx -180 ry 0 rz 90 deg; joints [74.155, -18.037, 85.889, 0, 22.148, 74.155]
  MoveL 2221 to (-21.28, 32.69, -3.5) mm, rotated rx -180 ry 0 rz 90 deg; joints [74.688, -18.236, 86.689, 0, 21.548, 74.688]
  MoveL 2222 to (-21.65, 33.7, -3.5) mm, rotated rx 180 ry 0 rz 90 deg; joints [74.717, -18.247, 86.734, 0, 21.514, 74.717]
  MoveC 2223 to (-22.86, 35.82, -3.5) mm, rotated rx 180 ry 0 rz 90 deg; joints [74.777, -18.278, 86.857, 0, 21.42, 74.777] to (-24.67, 37.44, -3.5) mm, rotated rx -180 ry 0 rz 90 deg; joints [74.814, -18.316, 87.014, 0, 21.302, 74.814]
  MoveL 2224 to (-66.81, 64.48, -3.5) mm, rotated rx 180 ry 0 rz 90 deg; joints [75.347, -19.095, 90.38, 0, 18.716, 75.347]
  MoveC 2225 to (-69.08, 65.63, -3.5) mm, rotated rx -180 ry 0 rz 90 deg; joints [75.365, -19.133, 90.552, 0, 18.581, 75.365] to (-71.55, 66.26, -3.5) mm, rotated rx 180 ry 0 rz 90 deg; joints [75.365, -19.171, 90.728, 0, 18.443, 75.365]
  MoveC 2226 to (-75.68, 65.37, -3.5) mm, rotated rx 180 ry 0 rz 90 deg; joints [75.297, -19.227, 90.988, 0, 18.239, 75.297] to (-78.32, 62.07, -3.5) mm, rotated rx 180 ry 0 rz 90 deg; joints [75.16, -19.252, 91.106, 0, 18.147, 75.16]
  MoveC 2227 to (-78.74, 60.41, -3.5) mm, rotated rx -180 ry 0 rz 90 deg; joints [75.099, -19.252, 91.105, 0, 18.148, 75.099] to (-78.88, 58.71, -3.5) mm, rotated rx -180 ry 0 rz 90 deg; joints [75.039, -19.248, 91.084, 0, 18.164, 75.039]
  MoveL 2228 to (-78.87, 29.38, -3.5) mm, rotated rx 180 ry 0 rz 90 deg; joints [74.036, -19.131, 90.544, 0, 18.588, 74.036]
  MoveL 2229 to (-71.33, 29.38, -3.5) mm, rotated rx -180 ry 0 rz 90 deg; joints [74.109, -19.021, 90.04, 0, 18.981, 74.109]
  MoveL 2230 to (-71.33, 29.38, -0.5) mm, rotated rx 180 ry 0 rz 90 deg; joints [74.109, -19.178, 90.141, 0, 19.037, 74.109]
  Establecer velocidad (1000.0 mm/s)
  MoveL 2231 to (-71.33, 29.38, 10) mm, rotated rx 180 ry 0 rz 90 deg; joints [74.109, -19.728, 90.49, 0, 19.237, 74.109]
  Establecer velocidad (66.7 mm/s)
  MoveL 2232 to (-70.64, -45.04, 10) mm, rotated rx -180 ry 0 rz 90 deg; joints [71.626, -19.362, 88.905, 0, 20.457, 71.626]
  MoveL 2233 to (-70.64, -45.04, -0.25) mm, rotated rx 180 ry 0 rz 90 deg; joints [71.626, -18.829, 88.564, 0, 20.265, 71.626]
  MoveL 2234 to (-72.14, -44.85, -0.66) mm, rotated rx 180 ry 0 rz 90 deg; joints [71.616, -18.832, 88.656, 0, 20.177, 71.616]
  MoveL 2235 to (-73.65, -45.04, -1.06) mm, rotated rx 180 ry 0 rz 90 deg; joints [71.593, -18.834, 88.739, 0, 20.095, 71.593]
  MoveL 2236 to (-75.08, -45.55, -1.47) mm, rotated rx -180 ry 0 rz 90 deg; joints [71.561, -18.832, 88.81, 0, 20.022, 71.561]
  MoveL 2237 to (-76.37, -46.37, -1.87) mm, rotated rx -180 ry 0 rz 90 deg; joints [71.519, -18.827, 88.864, 0, 19.963, 71.519]
  MoveL 2238 to (-77.43, -47.44, -2.28) mm, rotated rx -180 ry 0 rz 90 deg; joints [71.472, -18.817, 88.897, 0, 19.919, 71.472]
  MoveL 2239 to (-78.24, -48.73, -2.69) mm, rotated rx 180 ry 0 rz 90 deg; joints [71.42, -18.801, 88.909, 0, 19.892, 71.42]
  MoveL 2240 to (-78.74, -50.17, -3.09) mm, rotated rx -180 ry 0 rz 90 deg; joints [71.367, -18.78, 88.896, 0, 19.884, 71.367]
  MoveL 2241 to (-78.88, -51.68, -3.5) mm, rotated rx 180 ry 0 rz 90 deg; joints [71.316, -18.753, 88.858, 0, 19.896, 71.316]
  MoveL 2242 to (-78.88, -70.98, -3.5) mm, rotated rx 180 ry 0 rz 90 deg; joints [70.68, -18.65, 88.414, 0, 20.236, 70.68]
  MoveC 2243 to (-76.78, -76.08, -3.5) mm, rotated rx 180 ry 0 rz 90 deg; joints [70.538, -18.589, 88.154, 0, 20.436, 70.538] to (-71.7, -78.23, -3.5) mm, rotated rx -180 ry 0 rz 90 deg; joints [70.526, -18.496, 87.762, 0, 20.734, 70.526]
  MoveL 2244 to (-70.6, -78.24, -3.5) mm, rotated rx -180 ry 0 rz 90 deg; joints [70.538, -18.478, 87.687, 0, 20.791, 70.538]
  MoveL 2245 to (-35.54, -77.96, -3.5) mm, rotated rx 180 ry 0 rz 90 deg; joints [70.943, -17.889, 85.302, 0, 22.586, 70.943]
  MoveC 2246 to (-30.93, -76.48, -3.5) mm, rotated rx 180 ry 0 rz 90 deg; joints [71.041, -17.816, 85.018, 0, 22.797, 71.041] to (-28.2, -72.49, -3.5) mm, rotated rx -180 ry 0 rz 90 deg; joints [71.198, -17.791, 84.923, 0, 22.868, 71.198]
  MoveL 2247 to (-16.83, -28.9, -3.5) mm, rotated rx -180 ry 0 rz 90 deg; joints [72.718, -17.842, 85.121, 0, 22.721, 72.718]
  MoveL 2248 to (-15.53, -23.81, -3.5) mm, rotated rx 180 ry 0 rz 90 deg; joints [72.895, -17.847, 85.14, 0, 22.707, 72.895]
  MoveC 2249 to (-15.23, -21.6, -3.5) mm, rotated rx 180 ry 0 rz 90 deg; joints [72.97, -17.854, 85.167, 0, 22.687, 72.97] to (-15.46, -19.39, -3.5) mm, rotated rx 180 ry 0 rz 90 deg; joints [73.039, -17.87, 85.231, 0, 22.64, 73.039]
  MoveC 2250 to (-17.66, -15.89, -3.5) mm, rotated rx 180 ry 0 rz 90 deg; joints [73.131, -17.928, 85.459, 0, 22.47, 73.131] to (-21.57, -14.56, -3.5) mm, rotated rx 180 ry 0 rz 90 deg; joints [73.136, -18.005, 85.76, 0, 22.245, 73.136]
  MoveC 2251 to (-23.12, -14.65, -3.5) mm, rotated rx -180 ry 0 rz 90 deg; joints [73.117, -18.031, 85.866, 0, 22.165, 73.117] to (-24.66, -14.9, -3.5) mm, rotated rx -180 ry 0 rz 90 deg; joints [73.094, -18.057, 85.968, 0, 22.089, 73.094]
  MoveL 2252 to (-73.08, -25.21, -3.5) mm, rotated rx -180 ry 0 rz 90 deg; joints [72.257, -18.798, 89.052, 0, 19.746, 72.257]
  MoveC 2253 to (-77.25, -27.77, -3.5) mm, rotated rx 180 ry 0 rz 90 deg; joints [72.127, -18.849, 89.276, 0, 19.573, 72.127] to (-78.88, -32.38, -3.5) mm, rotated rx 180 ry 0 rz 90 deg; joints [71.956, -18.851, 89.285, 0, 19.566, 71.956]
  MoveL 2254 to (-78.88, -51.68, -3.5) mm, rotated rx 180 ry 0 rz 90 deg; joints [71.316, -18.753, 88.858, 0, 19.896, 71.316]
  MoveL 2255 to (-71.33, -51.68, -3.5) mm, rotated rx 180 ry 0 rz 90 deg; joints [71.4, -18.636, 88.352, 0, 20.284, 71.4]
  MoveL 2256 to (-71.33, -51.68, -0.5) mm, rotated rx 180 ry 0 rz 90 deg; joints [71.4, -18.792, 88.453, 0, 20.339, 71.4]
  Establecer velocidad (1000.0 mm/s)
  MoveL 2257 to (-71.33, -51.68, 10) mm, rotated rx -180 ry 0 rz 90 deg; joints [71.4, -19.337, 88.802, 0, 20.535, 71.4]
  Establecer velocidad (66.7 mm/s)
  MoveL 2258 to (18.39, -69.72, 10) mm, rotated rx 180 ry 0 rz 90 deg; joints [71.779, -17.606, 82.136, 0, 25.47, 71.779]
  MoveL 2259 to (18.39, -69.72, -0.25) mm, rotated rx -180 ry 0 rz 90 deg; joints [71.779, -17.089, 81.794, 0, 25.295, 71.779]
  MoveL 2260 to (18.22, -71.23, -0.66) mm, rotated rx 180 ry 0 rz 90 deg; joints [71.73, -17.061, 81.757, 0, 25.305, 71.73]
  MoveL 2261 to (18.42, -72.74, -1.06) mm, rotated rx 180 ry 0 rz 90 deg; joints [71.685, -17.027, 81.693, 0, 25.334, 71.685]
  MoveL 2262 to (18.95, -74.16, -1.47) mm, rotated rx 180 ry 0 rz 90 deg; joints [71.646, -16.986, 81.607, 0, 25.38, 71.646]
  MoveL 2263 to (19.77, -75.44, -1.87) mm, rotated rx 180 ry 0 rz 90 deg; joints [71.615, -16.94, 81.502, 0, 25.438, 71.615]
  MoveL 2264 to (20.86, -76.49, -2.28) mm, rotated rx -180 ry 0 rz 90 deg; joints [71.593, -16.891, 81.384, 0, 25.507, 71.593]
  MoveL 2265 to (22.16, -77.29, -2.69) mm, rotated rx 180 ry 0 rz 90 deg; joints [71.582, -16.838, 81.257, 0, 25.582, 71.582]
  MoveL 2266 to (23.6, -77.77, -3.09) mm, rotated rx 180 ry 0 rz 90 deg; joints [71.582, -16.785, 81.127, 0, 25.658, 71.582]
  MoveL 2267 to (25.11, -77.9, -3.5) mm, rotated rx 180 ry 0 rz 90 deg; joints [71.593, -16.733, 81, 0, 25.733, 71.593]
  MoveL 2268 to (46.91, -77.68, -3.5) mm, rotated rx -180 ry 0 rz 90 deg; joints [71.823, -16.276, 79.402, 0, 26.874, 71.823]
  MoveL 2269 to (53.54, -77.59, -3.5) mm, rotated rx -180 ry 0 rz 90 deg; joints [71.892, -16.133, 78.91, 0, 27.223, 71.892]
  MoveC 2270 to (54.7, -77.51, -3.5) mm, rotated rx -180 ry 0 rz 90 deg; joints [71.907, -16.108, 78.826, 0, 27.283, 71.907] to (55.84, -77.23, -3.5) mm, rotated rx 180 ry 0 rz 90 deg; joints [71.926, -16.085, 78.747, 0, 27.338, 71.926]
  MoveC 2271 to (58.74, -74, -3.5) mm, rotated rx 180 ry 0 rz 90 deg; joints [72.054, -16.045, 78.609, 0, 27.435, 72.054] to (58.86, -69.65, -3.5) mm, rotated rx 180 ry 0 rz 90 deg; joints [72.189, -16.073, 78.705, 0, 27.368, 72.189]
  MoveC 2272 to (58.14, -68.52, -3.5) mm, rotated rx 180 ry 0 rz 90 deg; joints [72.216, -16.097, 78.786, 0, 27.311, 72.216] to (57.32, -67.46, -3.5) mm, rotated rx -180 ry 0 rz 90 deg; joints [72.241, -16.122, 78.873, 0, 27.249, 72.241]
  MoveL 2273 to (29.71, -35.54, -3.5) mm, rotated rx -180 ry 0 rz 90 deg; joints [72.964, -16.915, 81.651, 0, 25.264, 72.964]
  MoveL 2274 to (27.99, -33.61, -3.5) mm, rotated rx -180 ry 0 rz 90 deg; joints [73.009, -16.961, 81.819, 0, 25.142, 73.009]
  MoveL 2275 to (27.01, -32.79, -3.5) mm, rotated rx 180 ry 0 rz 90 deg; joints [73.025, -16.986, 81.909, 0, 25.077, 73.025]
  MoveL 2276 to (13.25, -21.79, -3.5) mm, rotated rx -180 ry 0 rz 90 deg; joints [73.241, -17.323, 83.143, 0, 24.179, 73.241]
  MoveC 2277 to (11.68, -20.77, -3.5) mm, rotated rx 180 ry 0 rz 90 deg; joints [73.259, -17.359, 83.278, 0, 24.081, 73.259] to (9.94, -20.07, -3.5) mm, rotated rx -180 ry 0 rz 90 deg; joints [73.265, -17.396, 83.417, 0, 23.979, 73.265]
  MoveC 2278 to (6.44, -20.25, -3.5) mm, rotated rx 180 ry 0 rz 90 deg; joints [73.225, -17.462, 83.663, 0, 23.798, 73.225] to (3.82, -22.57, -3.5) mm, rotated rx -180 ry 0 rz 90 deg; joints [73.126, -17.498, 83.8, 0, 23.698, 73.126]
  MoveC 2279 to (3.26, -23.75, -3.5) mm, rotated rx 180 ry 0 rz 90 deg; joints [73.082, -17.502, 83.815, 0, 23.687, 73.082] to (2.84, -24.99, -3.5) mm, rotated rx 180 ry 0 rz 90 deg; joints [73.038, -17.502, 83.817, 0, 23.685, 73.038]
  MoveL 2280 to (-9.27, -70.6, -3.5) mm, rotated rx -180 ry 0 rz 90 deg; joints [71.462, -17.456, 83.641, 0, 23.815, 71.462]
  MoveC 2281 to (-9.3, -73.62, -3.5) mm, rotated rx 180 ry 0 rz 90 deg; joints [71.366, -17.437, 83.572, 0, 23.866, 71.366] to (-7.87, -76.29, -3.5) mm, rotated rx 180 ry 0 rz 90 deg; joints [71.297, -17.393, 83.406, 0, 23.987, 71.297]
  MoveC 2282 to (-5.76, -77.63, -3.5) mm, rotated rx -180 ry 0 rz 90 deg; joints [71.277, -17.345, 83.225, 0, 24.12, 71.277] to (-3.32, -78.14, -3.5) mm, rotated rx 180 ry 0 rz 90 deg; joints [71.287, -17.295, 83.039, 0, 24.255, 71.287]
  MoveL 2283 to (-2.37, -78.16, -3.5) mm, rotated rx 180 ry 0 rz 90 deg; joints [71.297, -17.276, 82.971, 0, 24.305, 71.297]
  MoveL 2284 to (25.11, -77.9, -3.5) mm, rotated rx 180 ry 0 rz 90 deg; joints [71.593, -16.733, 81, 0, 25.733, 71.593]
  MoveL 2285 to (25.04, -70.35, -3.5) mm, rotated rx -180 ry 0 rz 90 deg; joints [71.828, -16.785, 81.187, 0, 25.599, 71.828]
  MoveL 2286 to (25.04, -70.35, -0.5) mm, rotated rx 180 ry 0 rz 90 deg; joints [71.828, -16.937, 81.288, 0, 25.649, 71.828]
  Establecer velocidad (1000.0 mm/s)
  MoveL 2287 to (25.04, -70.35, 10) mm, rotated rx 180 ry 0 rz 90 deg; joints [71.828, -17.467, 81.639, 0, 25.827, 71.828]
  Establecer velocidad (66.7 mm/s)
  MoveL 2288 to (68.18, -31.22, 10) mm, rotated rx 180 ry 0 rz 90 deg; joints [73.461, -16.805, 79.352, 0, 27.453, 73.461]
  MoveL 2289 to (68.18, -31.22, -0.25) mm, rotated rx 180 ry 0 rz 90 deg; joints [73.461, -16.292, 79.008, 0, 27.284, 73.461]
  MoveL 2290 to (69.68, -31.4, -0.66) mm, rotated rx -180 ry 0 rz 90 deg; joints [73.469, -16.237, 78.877, 0, 27.361, 73.469]
  MoveL 2291 to (71.19, -31.22, -1.06) mm, rotated rx -180 ry 0 rz 90 deg; joints [73.489, -16.185, 78.753, 0, 27.431, 73.489]
  MoveL 2292 to (72.62, -30.71, -1.47) mm, rotated rx 180 ry 0 rz 90 deg; joints [73.518, -16.136, 78.643, 0, 27.493, 73.518]
  MoveL 2293 to (73.9, -29.89, -1.87) mm, rotated rx 180 ry 0 rz 90 deg; joints [73.554, -16.092, 78.55, 0, 27.542, 73.554]
  MoveL 2294 to (74.97, -28.81, -2.28) mm, rotated rx 180 ry 0 rz 90 deg; joints [73.597, -16.055, 78.479, 0, 27.576, 73.597]
  MoveL 2295 to (75.78, -27.52, -2.69) mm, rotated rx 180 ry 0 rz 90 deg; joints [73.644, -16.025, 78.433, 0, 27.592, 73.644]
  MoveL 2296 to (76.28, -26.09, -3.09) mm, rotated rx 180 ry 0 rz 90 deg; joints [73.693, -16.003, 78.413, 0, 27.59, 73.693]
  MoveL 2297 to (76.42, -24.58, -3.5) mm, rotated rx 180 ry 0 rz 90 deg; joints [73.741, -15.989, 78.422, 0, 27.567, 73.741]
  MoveL 2298 to (76.42, -5.21, -3.5) mm, rotated rx 180 ry 0 rz 90 deg; joints [74.341, -16.113, 78.842, 0, 27.271, 74.341]
  MoveL 2299 to (76.41, -4.26, -3.5) mm, rotated rx 180 ry 0 rz 90 deg; joints [74.37, -16.119, 78.863, 0, 27.256, 74.37]
  MoveL 2300 to (76.38, -3.79, -3.5) mm, rotated rx 180 ry 0 rz 90 deg; joints [74.384, -16.123, 78.875, 0, 27.248, 74.384]
  MoveC 2301 to (76.08, -2.51, -3.5) mm, rotated rx -180 ry 0 rz 90 deg; joints [74.422, -16.137, 78.925, 0, 27.212, 74.422] to (75.33, -1.42, -3.5) mm, rotated rx -180 ry 0 rz 90 deg; joints [74.449, -16.161, 79.005, 0, 27.156, 74.449]
  MoveC 2302 to (71.81, 1.05, -3.5) mm, rotated rx 180 ry 0 rz 90 deg; joints [74.496, -16.253, 79.323, 0, 26.931, 74.496] to (67.52, 0.7, -3.5) mm, rotated rx 180 ry 0 rz 90 deg; joints [74.447, -16.345, 79.638, 0, 26.707, 74.447]
  MoveL 2303 to (67.3, 0.47, -3.5) mm, rotated rx 180 ry 0 rz 90 deg; joints [74.438, -16.348, 79.65, 0, 26.698, 74.438]
  MoveL 2304 to (63.78, -4.26, -3.5) mm, rotated rx 180 ry 0 rz 90 deg; joints [74.259, -16.395, 79.814, 0, 26.581, 74.259]
  MoveL 2305 to (50.66, -22.27, -3.5) mm, rotated rx 180 ry 0 rz 90 deg; joints [73.578, -16.564, 80.405, 0, 26.16, 73.578]
  MoveL 2306 to (50.13, -23.03, -3.5) mm, rotated rx 180 ry 0 rz 90 deg; joints [73.549, -16.571, 80.427, 0, 26.144, 73.549]
  MoveC 2307 to (49.2, -26.39, -3.5) mm, rotated rx -180 ry 0 rz 90 deg; joints [73.436, -16.569, 80.422, 0, 26.147, 73.436] to (50.53, -29.61, -3.5) mm, rotated rx -180 ry 0 rz 90 deg; joints [73.348, -16.521, 80.252, 0, 26.269, 73.348]
  MoveL 2308 to (66.69, -47.86, -3.5) mm, rotated rx -180 ry 0 rz 90 deg; joints [72.934, -16.051, 78.631, 0, 27.42, 72.934]
  MoveL 2309 to (66.81, -47.99, -3.5) mm, rotated rx 180 ry 0 rz 90 deg; joints [72.931, -16.047, 78.619, 0, 27.429, 72.931]
  MoveL 2310 to (67.57, -48.8, -3.5) mm, rotated rx 180 ry 0 rz 90 deg; joints [72.913, -16.025, 78.542, 0, 27.483, 72.913]
  MoveC 2311 to (68.53, -49.44, -3.5) mm, rotated rx 180 ry 0 rz 90 deg; joints [72.903, -15.999, 78.456, 0, 27.544, 72.903] to (69.65, -49.66, -3.5) mm, rotated rx -180 ry 0 rz 90 deg; joints [72.906, -15.973, 78.365, 0, 27.607, 72.906]
  MoveL 2312 to (69.88, -49.67, -3.5) mm, rotated rx -180 ry 0 rz 90 deg; joints [72.908, -15.967, 78.348, 0, 27.62, 72.908]
  MoveC 2313 to (73.74, -48.49, -3.5) mm, rotated rx -180 ry 0 rz 90 deg; joints [72.981, -15.889, 78.083, 0, 27.806, 72.981] to (76.29, -45.36, -3.5) mm, rotated rx 180 ry 0 rz 90 deg; joints [73.101, -15.853, 77.962, 0, 27.891, 73.101]
  MoveL 2314 to (76.35, -45.01, -3.5) mm, rotated rx 180 ry 0 rz 90 deg; joints [73.112, -15.854, 77.965, 0, 27.889, 73.112]
  MoveL 2315 to (76.42, -43.12, -3.5) mm, rotated rx -180 ry 0 rz 90 deg; joints [73.171, -15.866, 78.004, 0, 27.862, 73.171]
  MoveL 2316 to (76.42, -24.58, -3.5) mm, rotated rx 180 ry 0 rz 90 deg; joints [73.741, -15.989, 78.422, 0, 27.567, 73.741]
  MoveL 2317 to (68.86, -24.58, -3.5) mm, rotated rx 180 ry 0 rz 90 deg; joints [73.673, -16.157, 78.993, 0, 27.164, 73.673]
  MoveL 2318 to (68.86, -24.58, -0.5) mm, rotated rx -180 ry 0 rz 90 deg; joints [73.673, -16.308, 79.095, 0, 27.212, 73.673]
  Establecer velocidad (1000.0 mm/s)
  MoveL 2319 to (68.86, -24.58, 10) mm, rotated rx -180 ry 0 rz 90 deg; joints [73.673, -16.833, 79.448, 0, 27.386, 73.673]
  Establecer velocidad (66.7 mm/s)
  MoveL 2320 to (36.72, 8.05, 10) mm, rotated rx 180 ry 0 rz 90 deg; joints [74.408, -17.714, 82.522, 0, 25.192, 74.408]
  MoveL 2321 to (36.72, 8.05, -0.25) mm, rotated rx 180 ry 0 rz 90 deg; joints [74.408, -17.195, 82.18, 0, 25.015, 74.408]
  MoveL 2322 to (37.84, 7.02, -0.66) mm, rotated rx 180 ry 0 rz 90 deg; joints [74.386, -17.147, 82.064, 0, 25.083, 74.386]
  MoveL 2323 to (39.17, 6.29, -1.06) mm, rotated rx -180 ry 0 rz 90 deg; joints [74.374, -17.095, 81.938, 0, 25.157, 74.374]
  MoveL 2324 to (40.63, 5.87, -1.47) mm, rotated rx 180 ry 0 rz 90 deg; joints [74.374, -17.042, 81.808, 0, 25.234, 74.374]
  MoveL 2325 to (42.15, 5.79, -1.87) mm, rotated rx -180 ry 0 rz 90 deg; joints [74.385, -16.99, 81.682, 0, 25.309, 74.385]
  MoveL 2326 to (43.64, 6.04, -2.28) mm, rotated rx 180 ry 0 rz 90 deg; joints [74.406, -16.941, 81.563, 0, 25.377, 74.406]
  MoveL 2327 to (45.05, 6.62, -2.69) mm, rotated rx 180 ry 0 rz 90 deg; joints [74.437, -16.895, 81.458, 0, 25.437, 74.437]
  MoveL 2328 to (46.29, 7.5, -3.09) mm, rotated rx 180 ry 0 rz 90 deg; joints [74.475, -16.853, 81.371, 0, 25.483, 74.475]
  MoveL 2329 to (47.28, 8.64, -3.5) mm, rotated rx 180 ry 0 rz 90 deg; joints [74.52, -16.819, 81.307, 0, 25.512, 74.52]
  MoveL 2330 to (58.43, 24.17, -3.5) mm, rotated rx 180 ry 0 rz 90 deg; joints [75.107, -16.675, 80.794, 0, 25.881, 75.107]
  MoveL 2331 to (59.21, 25.32, -3.5) mm, rotated rx 180 ry 0 rz 90 deg; joints [75.15, -16.665, 80.759, 0, 25.906, 75.15]
  MoveC 2332 to (60.14, 28.33, -3.5) mm, rotated rx 180 ry 0 rz 90 deg; joints [75.253, -16.662, 80.749, 0, 25.913, 75.253] to (59.23, 31.36, -3.5) mm, rotated rx 180 ry 0 rz 90 deg; joints [75.341, -16.698, 80.876, 0, 25.822, 75.341]
  MoveC 2333 to (57.38, 33.41, -3.5) mm, rotated rx 180 ry 0 rz 90 deg; joints [75.391, -16.748, 81.053, 0, 25.695, 75.391] to (54.72, 34.15, -3.5) mm, rotated rx 180 ry 0 rz 90 deg; joints [75.392, -16.807, 81.264, 0, 25.543, 75.392]
  MoveL 2334 to (53.54, 34.13, -3.5) mm, rotated rx -180 ry 0 rz 90 deg; joints [75.382, -16.831, 81.351, 0, 25.48, 75.382]
  MoveL 2335 to (8.05, 32.91, -3.5) mm, rotated rx -180 ry 0 rz 90 deg; joints [74.955, -17.715, 84.629, 0, 23.087, 74.955]
  MoveL 2336 to (7.11, 32.83, -3.5) mm, rotated rx -180 ry 0 rz 90 deg; joints [74.945, -17.732, 84.695, 0, 23.038, 74.945]
  MoveC 2337 to (4.93, 32.29, -3.5) mm, rotated rx -180 ry 0 rz 90 deg; joints [74.908, -17.77, 84.839, 0, 22.931, 74.908] to (3.02, 31.1, -3.5) mm, rotated rx -180 ry 0 rz 90 deg; joints [74.853, -17.799, 84.952, 0, 22.847, 74.853]
  MoveC 2338 to (1.57, 28.28, -3.5) mm, rotated rx 180 ry 0 rz 90 deg; joints [74.748, -17.811, 85, 0, 22.811, 74.748] to (1.8, 25.11, -3.5) mm, rotated rx 180 ry 0 rz 90 deg; joints [74.646, -17.791, 84.922, 0, 22.869, 74.646]
  MoveL 2339 to (2.11, 24.17, -3.5) mm, rotated rx -180 ry 0 rz 90 deg; joints [74.618, -17.781, 84.882, 0, 22.899, 74.618]
  MoveL 2340 to (8.08, 7.73, -3.5) mm, rotated rx 180 ry 0 rz 90 deg; joints [74.14, -17.585, 84.13, 0, 23.455, 74.14]
  MoveC 2341 to (8.87, 6.25, -3.5) mm, rotated rx 180 ry 0 rz 90 deg; joints [74.099, -17.562, 84.044, 0, 23.518, 74.099] to (10.03, 5.05, -3.5) mm, rotated rx 180 ry 0 rz 90 deg; joints [74.071, -17.534, 83.937, 0, 23.597, 74.071]
  MoveL 2342 to (27.01, -8.17, -3.5) mm, rotated rx 180 ry 0 rz 90 deg; joints [73.805, -17.132, 82.441, 0, 24.691, 73.805]
  MoveL 2343 to (27.78, -8.72, -3.5) mm, rotated rx 180 ry 0 rz 90 deg; joints [73.794, -17.114, 82.373, 0, 24.741, 73.794]
  MoveC 2344 to (31.66, -9.75, -3.5) mm, rotated rx -180 ry 0 rz 90 deg; joints [73.797, -17.031, 82.07, 0, 24.961, 73.797] to (35.24, -7.94, -3.5) mm, rotated rx -180 ry 0 rz 90 deg; joints [73.888, -16.969, 81.847, 0, 25.122, 73.888]
  MoveL 2345 to (35.54, -7.62, -3.5) mm, rotated rx -180 ry 0 rz 90 deg; joints [73.901, -16.965, 81.832, 0, 25.133, 73.901]
  MoveL 2346 to (35.97, -7.11, -3.5) mm, rotated rx 180 ry 0 rz 90 deg; joints [73.921, -16.959, 81.811, 0, 25.148, 73.921]
  MoveL 2347 to (42.17, 1.51, -3.5) mm, rotated rx 180 ry 0 rz 90 deg; joints [74.249, -16.883, 81.537, 0, 25.346, 74.249]
  MoveL 2348 to (47.28, 8.64, -3.5) mm, rotated rx 180 ry 0 rz 90 deg; joints [74.52, -16.819, 81.307, 0, 25.512, 74.52]
  MoveL 2349 to (41.15, 13.04, -3.5) mm, rotated rx -180 ry 0 rz 90 deg; joints [74.606, -16.969, 81.847, 0, 25.122, 74.606]
  MoveL 2350 to (41.15, 13.04, -0.5) mm, rotated rx -180 ry 0 rz 90 deg; joints [74.606, -17.121, 81.949, 0, 25.172, 74.606]
  Establecer velocidad (1000.0 mm/s)
  MoveL 2351 to (41.15, 13.04, 10) mm, rotated rx -180 ry 0 rz 90 deg; joints [74.606, -17.652, 82.299, 0, 25.353, 74.606]
  Establecer velocidad (66.7 mm/s)
  MoveL 2352 to (24.44, 69.5, 10) mm, rotated rx 180 ry 0 rz 90 deg; joints [76.284, -18.273, 84.577, 0, 23.696, 76.284]
  MoveL 2353 to (24.44, 69.5, -0.25) mm, rotated rx -180 ry 0 rz 90 deg; joints [76.284, -17.75, 84.236, 0, 23.514, 76.284]
  MoveL 2354 to (24.65, 71, -0.66) mm, rotated rx 180 ry 0 rz 90 deg; joints [76.334, -17.732, 84.234, 0, 23.498, 76.334]
  MoveL 2355 to (24.48, 72.51, -1.06) mm, rotated rx 180 ry 0 rz 90 deg; joints [76.382, -17.722, 84.259, 0, 23.463, 76.382]
  MoveL 2356 to (23.99, 73.95, -1.47) mm, rotated rx -180 ry 0 rz 90 deg; joints [76.425, -17.717, 84.306, 0, 23.411, 76.425]
  MoveL 2357 to (23.19, 75.24, -1.87) mm, rotated rx 180 ry 0 rz 90 deg; joints [76.461, -17.717, 84.372, 0, 23.345, 76.461]
  MoveL 2358 to (22.12, 76.32, -2.28) mm, rotated rx 180 ry 0 rz 90 deg; joints [76.488, -17.721, 84.454, 0, 23.267, 76.488]
  MoveL 2359 to (20.84, 77.14, -2.69) mm, rotated rx -180 ry 0 rz 90 deg; joints [76.505, -17.728, 84.546, 0, 23.182, 76.505]
  MoveL 2360 to (19.41, 77.65, -3.09) mm, rotated rx -180 ry 0 rz 90 deg; joints [76.51, -17.736, 84.644, 0, 23.092, 76.51]
  MoveL 2361 to (17.9, 77.81, -3.5) mm, rotated rx -180 ry 0 rz 90 deg; joints [76.504, -17.744, 84.741, 0, 23.003, 76.504]
  MoveC 2362 to (15.06, 77.84, -3.5) mm, rotated rx -180 ry 0 rz 90 deg; joints [76.482, -17.797, 84.945, 0, 22.852, 76.482] to (12.22, 77.87, -3.5) mm, rotated rx -180 ry 0 rz 90 deg; joints [76.461, -17.849, 85.148, 0, 22.701, 76.461]
  MoveL 2363 to (-29.85, 78.29, -3.5) mm, rotated rx -180 ry 0 rz 90 deg; joints [76.134, -18.577, 88.104, 0, 20.473, 76.134]
  MoveC 2364 to (-32.71, 78.17, -3.5) mm, rotated rx 180 ry 0 rz 90 deg; joints [76.106, -18.623, 88.299, 0, 20.324, 76.106] to (-35.54, 77.75, -3.5) mm, rotated rx 180 ry 0 rz 90 deg; joints [76.068, -18.667, 88.486, 0, 20.181, 76.068]
  MoveC 2365 to (-38.77, 73.93, -3.5) mm, rotated rx -180 ry 0 rz 90 deg; joints [75.912, -18.704, 88.643, 0, 20.061, 75.912] to (-38.13, 68.97, -3.5) mm, rotated rx 180 ry 0 rz 90 deg; joints [75.75, -18.673, 88.513, 0, 20.161, 75.75]
  MoveC 2366 to (-36.88, 67.89, -3.5) mm, rotated rx -180 ry 0 rz 90 deg; joints [75.724, -18.649, 88.409, 0, 20.24, 75.724] to (-35.54, 66.94, -3.5) mm, rotated rx 180 ry 0 rz 90 deg; joints [75.704, -18.623, 88.3, 0, 20.324, 75.704]
  MoveL 2367 to (-12.46, 52.31, -3.5) mm, rotated rx -180 ry 0 rz 90 deg; joints [75.414, -18.175, 86.439, 0, 21.735, 75.414]
  MoveC 2368 to (-9.76, 51.15, -3.5) mm, rotated rx -180 ry 0 rz 90 deg; joints [75.399, -18.122, 86.228, 0, 21.894, 75.399] to (-6.82, 50.9, -3.5) mm, rotated rx -180 ry 0 rz 90 deg; joints [75.416, -18.07, 86.018, 0, 22.052, 75.416]
  MoveC 2369 to (32.34, 53.77, -3.5) mm, rotated rx -180 ry 0 rz 90 deg; joints [75.837, -17.358, 83.274, 0, 24.084, 75.837] to (71.5, 56.55, -3.5) mm, rotated rx 180 ry 0 rz 90 deg; joints [76.238, -16.573, 80.436, 0, 26.138, 76.238]
  MoveC 2370 to (74.68, 58.06, -3.5) mm, rotated rx 180 ry 0 rz 90 deg; joints [76.31, -16.513, 80.225, 0, 26.289, 76.31] to (75.98, 61.33, -3.5) mm, rotated rx 180 ry 0 rz 90 deg; joints [76.423, -16.502, 80.186, 0, 26.316, 76.423]
  MoveL 2371 to (75.99, 62.07, -3.5) mm, rotated rx 180 ry 0 rz 90 deg; joints [76.447, -16.506, 80.199, 0, 26.307, 76.447]
  MoveL 2372 to (75.99, 71.55, -3.5) mm, rotated rx 180 ry 0 rz 90 deg; joints [76.747, -16.554, 80.369, 0, 26.185, 76.747]
  MoveL 2373 to (75.98, 72.21, -3.5) mm, rotated rx -180 ry 0 rz 90 deg; joints [76.768, -16.558, 80.382, 0, 26.176, 76.768]
  MoveC 2374 to (74.6, 75.45, -3.5) mm, rotated rx 180 ry 0 rz 90 deg; joints [76.861, -16.603, 80.542, 0, 26.061, 76.861] to (71.37, 76.85, -3.5) mm, rotated rx 180 ry 0 rz 90 deg; joints [76.881, -16.679, 80.809, 0, 25.87, 76.881]
  MoveC 2375 to (44.63, 77.42, -3.5) mm, rotated rx 180 ry 0 rz 90 deg; joints [76.698, -17.23, 82.799, 0, 24.431, 76.698] to (17.9, 77.81, -3.5) mm, rotated rx -180 ry 0 rz 90 deg; joints [76.504, -17.744, 84.741, 0, 23.003, 76.504]
  MoveL 2376 to (17.82, 70.26, -3.5) mm, rotated rx 180 ry 0 rz 90 deg; joints [76.256, -17.712, 84.616, 0, 23.096, 76.256]
  MoveL 2377 to (17.82, 70.26, -0.5) mm, rotated rx -180 ry 0 rz 90 deg; joints [76.256, -17.865, 84.717, 0, 23.148, 76.256]
  Establecer velocidad (1000.0 mm/s)
  MoveL 2378 to (17.82, 70.26, 10) mm, rotated rx 180 ry 0 rz 90 deg; joints [76.256, -18.402, 85.066, 0, 23.336, 76.256]
  Establecer velocidad (66.7 mm/s)
  MoveL 2379 to (24.44, 69.17, 10) mm, rotated rx -180 ry 0 rz 90 deg; joints [76.273, -18.271, 84.571, 0, 23.7, 76.273]
  MoveL 2380 to (24.44, 69.17, -0.5) mm, rotated rx 180 ry 0 rz 90 deg; joints [76.273, -17.736, 84.222, 0, 23.514, 76.273]
  MoveL 2381 to (24.65, 70.67, -0.91) mm, rotated rx 180 ry 0 rz 90 deg; joints [76.324, -17.718, 84.22, 0, 23.498, 76.324]
  MoveL 2382 to (24.48, 72.18, -1.31) mm, rotated rx 180 ry 0 rz 90 deg; joints [76.372, -17.707, 84.245, 0, 23.463, 76.372]
  MoveL 2383 to (23.99, 73.62, -1.72) mm, rotated rx -180 ry 0 rz 90 deg; joints [76.415, -17.703, 84.292, 0, 23.411, 76.415]
  MoveL 2384 to (23.19, 74.91, -2.13) mm, rotated rx 180 ry 0 rz 90 deg; joints [76.451, -17.703, 84.358, 0, 23.345, 76.451]
  MoveL 2385 to (22.12, 76, -2.53) mm, rotated rx 180 ry 0 rz 90 deg; joints [76.478, -17.707, 84.44, 0, 23.267, 76.478]
  MoveL 2386 to (20.84, 76.82, -2.94) mm, rotated rx 180 ry 0 rz 90 deg; joints [76.494, -17.714, 84.533, 0, 23.181, 76.494]
  MoveL 2387 to (19.41, 77.34, -3.34) mm, rotated rx 180 ry 0 rz 90 deg; joints [76.5, -17.722, 84.63, 0, 23.092, 76.5]
  MoveL 2388 to (17.9, 77.49, -3.75) mm, rotated rx 180 ry 0 rz 90 deg; joints [76.493, -17.73, 84.727, 0, 23.003, 76.493]
  MoveC 2389 to (13.45, 77.54, -3.75) mm, rotated rx -180 ry 0 rz 90 deg; joints [76.46, -17.812, 85.046, 0, 22.766, 76.46] to (9, 77.58, -3.75) mm, rotated rx 180 ry 0 rz 90 deg; joints [76.426, -17.894, 85.364, 0, 22.53, 76.426]
  MoveL 2390 to (-28.9, 77.97, -3.75) mm, rotated rx -180 ry 0 rz 90 deg; joints [76.131, -18.548, 88.025, 0, 20.523, 76.131]
  MoveL 2391 to (-30.44, 77.97, -3.75) mm, rotated rx 180 ry 0 rz 90 deg; joints [76.118, -18.573, 88.131, 0, 20.442, 76.118]
  MoveC 2392 to (-32.76, 77.86, -3.75) mm, rotated rx -180 ry 0 rz 90 deg; joints [76.095, -18.61, 88.289, 0, 20.321, 76.095] to (-35.05, 77.49, -3.75) mm, rotated rx -180 ry 0 rz 90 deg; joints [76.063, -18.645, 88.44, 0, 20.205, 76.063]
  MoveC 2393 to (-38.16, 73.66, -3.75) mm, rotated rx -180 ry 0 rz 90 deg; joints [75.908, -18.68, 88.588, 0, 20.092, 75.908] to (-37.43, 68.77, -3.75) mm, rotated rx -180 ry 0 rz 90 deg; joints [75.749, -18.648, 88.453, 0, 20.195, 75.749]
  MoveL 2394 to (-36.91, 68.3, -3.75) mm, rotated rx 180 ry 0 rz 90 deg; joints [75.738, -18.638, 88.409, 0, 20.229, 75.738]
  MoveL 2395 to (-33.64, 66.11, -3.75) mm, rotated rx 180 ry 0 rz 90 deg; joints [75.692, -18.576, 88.147, 0, 20.43, 75.692]
  MoveL 2396 to (-12.33, 52.6, -3.75) mm, rotated rx 180 ry 0 rz 90 deg; joints [75.425, -18.161, 86.427, 0, 21.734, 75.425]
  MoveC 2397 to (-9.71, 51.47, -3.75) mm, rotated rx -180 ry 0 rz 90 deg; joints [75.41, -18.11, 86.222, 0, 21.888, 75.41] to (-6.86, 51.23, -3.75) mm, rotated rx 180 ry 0 rz 90 deg; joints [75.426, -18.059, 86.018, 0, 22.041, 75.426]
  MoveC 2398 to (32.22, 54.09, -3.75) mm, rotated rx 180 ry 0 rz 90 deg; joints [75.846, -17.349, 83.28, 0, 24.069, 75.846] to (71.3, 56.88, -3.75) mm, rotated rx -180 ry 0 rz 90 deg; joints [76.246, -16.567, 80.448, 0, 26.119, 76.246]
  MoveC 2399 to (74.38, 58.34, -3.75) mm, rotated rx 180 ry 0 rz 90 deg; joints [76.316, -16.508, 80.244, 0, 26.265, 76.316] to (75.65, 61.49, -3.75) mm, rotated rx -180 ry 0 rz 90 deg; joints [76.426, -16.498, 80.206, 0, 26.292, 76.426]
  MoveL 2400 to (75.65, 62.07, -3.75) mm, rotated rx 180 ry 0 rz 90 deg; joints [76.444, -16.5, 80.216, 0, 26.285, 76.444]
  MoveL 2401 to (75.65, 71.92, -3.75) mm, rotated rx -180 ry 0 rz 90 deg; joints [76.757, -16.551, 80.392, 0, 26.158, 76.757]
  MoveC 2402 to (74.35, 75.13, -3.75) mm, rotated rx 180 ry 0 rz 90 deg; joints [76.849, -16.595, 80.547, 0, 26.048, 76.849] to (71.17, 76.52, -3.75) mm, rotated rx 180 ry 0 rz 90 deg; joints [76.869, -16.669, 80.81, 0, 25.859, 76.869]
  MoveC 2403 to (44.53, 77.09, -3.75) mm, rotated rx 180 ry 0 rz 90 deg; joints [76.687, -17.217, 82.792, 0, 24.425, 76.687] to (17.9, 77.49, -3.75) mm, rotated rx 180 ry 0 rz 90 deg; joints [76.493, -17.73, 84.727, 0, 23.003, 76.493]
  MoveL 2404 to (17.81, 69.94, -3.75) mm, rotated rx 180 ry 0 rz 90 deg; joints [76.245, -17.698, 84.602, 0, 23.095, 76.245]
  MoveL 2405 to (17.81, 69.94, -0.75) mm, rotated rx -180 ry 0 rz 90 deg; joints [76.245, -17.851, 84.703, 0, 23.148, 76.245]
  Establecer velocidad (1000.0 mm/s)
  MoveL 2406 to (17.81, 69.94, 10) mm, rotated rx 180 ry 0 rz 90 deg; joints [76.245, -18.401, 85.061, 0, 23.339, 76.245]
  Establecer velocidad (66.7 mm/s)
  MoveL 2407 to (38.03, 25.13, 10) mm, rotated rx -180 ry 0 rz 90 deg; joints [74.964, -17.782, 82.768, 0, 25.015, 74.964]
  MoveL 2408 to (38.03, 25.13, -0.5) mm, rotated rx -180 ry 0 rz 90 deg; joints [74.964, -17.25, 82.417, 0, 24.833, 74.964]
  MoveL 2409 to (38.18, 26.64, -0.91) mm, rotated rx -180 ry 0 rz 90 deg; joints [75.014, -17.235, 82.423, 0, 24.812, 75.014]
  MoveL 2410 to (37.96, 28.14, -1.31) mm, rotated rx 180 ry 0 rz 90 deg; joints [75.06, -17.227, 82.455, 0, 24.772, 75.06]
  MoveL 2411 to (37.4, 29.56, -1.72) mm, rotated rx -180 ry 0 rz 90 deg; joints [75.101, -17.225, 82.509, 0, 24.716, 75.101]
  MoveL 2412 to (36.56, 30.82, -2.13) mm, rotated rx 180 ry 0 rz 90 deg; joints [75.134, -17.228, 82.581, 0, 24.646, 75.134]
  MoveL 2413 to (35.45, 31.86, -2.53) mm, rotated rx -180 ry 0 rz 90 deg; joints [75.158, -17.235, 82.668, 0, 24.566, 75.158]
  MoveL 2414 to (34.14, 32.63, -2.94) mm, rotated rx 180 ry 0 rz 90 deg; joints [75.171, -17.244, 82.765, 0, 24.479, 75.171]
  MoveL 2415 to (32.69, 33.09, -3.34) mm, rotated rx 180 ry 0 rz 90 deg; joints [75.174, -17.254, 82.865, 0, 24.389, 75.174]
  MoveL 2416 to (31.18, 33.19, -3.75) mm, rotated rx -180 ry 0 rz 90 deg; joints [75.164, -17.264, 82.963, 0, 24.3, 75.164]
  MoveL 2417 to (7.6, 32.56, -3.75) mm, rotated rx 180 ry 0 rz 90 deg; joints [74.94, -17.709, 84.646, 0, 23.063, 74.94]
  MoveC 2418 to (5.6, 32.2, -3.75) mm, rotated rx -180 ry 0 rz 90 deg; joints [74.911, -17.744, 84.781, 0, 22.963, 74.911] to (3.79, 31.26, -3.75) mm, rotated rx -180 ry 0 rz 90 deg; joints [74.864, -17.773, 84.892, 0, 22.881, 74.864]
  MoveC 2419 to (2.05, 28.93, -3.75) mm, rotated rx 180 ry 0 rz 90 deg; joints [74.773, -17.793, 84.971, 0, 22.822, 74.773] to (1.91, 26.03, -3.75) mm, rotated rx -180 ry 0 rz 90 deg; joints [74.677, -17.781, 84.924, 0, 22.857, 74.677]
  MoveL 2420 to (2.15, 25.11, -3.75) mm, rotated rx -180 ry 0 rz 90 deg; joints [74.65, -17.772, 84.89, 0, 22.883, 74.65]
  MoveL 2421 to (2.47, 24.17, -3.75) mm, rotated rx 180 ry 0 rz 90 deg; joints [74.622, -17.761, 84.848, 0, 22.913, 74.622]
  MoveL 2422 to (8.36, 7.93, -3.75) mm, rotated rx 180 ry 0 rz 90 deg; joints [74.149, -17.568, 84.107, 0, 23.462, 74.149]
  MoveC 2423 to (9.14, 6.45, -3.75) mm, rotated rx 180 ry 0 rz 90 deg; joints [74.108, -17.546, 84.02, 0, 23.525, 74.108] to (10.31, 5.24, -3.75) mm, rotated rx -180 ry 0 rz 90 deg; joints [74.08, -17.517, 83.913, 0, 23.604, 74.08]
  MoveL 2424 to (27.75, -8.32, -3.75) mm, rotated rx 180 ry 0 rz 90 deg; joints [73.807, -17.104, 82.376, 0, 24.728, 73.807]
  MoveC 2425 to (31.5, -9.43, -3.75) mm, rotated rx -180 ry 0 rz 90 deg; joints [73.806, -17.023, 82.08, 0, 24.943, 73.806] to (35.01, -7.7, -3.75) mm, rotated rx 180 ry 0 rz 90 deg; joints [73.893, -16.963, 81.86, 0, 25.102, 73.893]
  MoveL 2426 to (35.55, -7.11, -3.75) mm, rotated rx 180 ry 0 rz 90 deg; joints [73.917, -16.955, 81.833, 0, 25.122, 73.917]
  MoveL 2427 to (38.38, -3.22, -3.75) mm, rotated rx -180 ry 0 rz 90 deg; joints [74.066, -16.92, 81.708, 0, 25.212, 74.066]
  MoveL 2428 to (56.67, 22.27, -3.75) mm, rotated rx -180 ry 0 rz 90 deg; joints [75.032, -16.689, 80.879, 0, 25.81, 75.032]
  MoveL 2429 to (58.86, 25.35, -3.75) mm, rotated rx 180 ry 0 rz 90 deg; joints [75.148, -16.66, 80.777, 0, 25.883, 75.148]
  MoveC 2430 to (59.49, 26.68, -3.75) mm, rotated rx 180 ry 0 rz 90 deg; joints [75.195, -16.654, 80.756, 0, 25.898, 75.195] to (59.62, 28.16, -3.75) mm, rotated rx 180 ry 0 rz 90 deg; joints [75.243, -16.659, 80.776, 0, 25.884, 75.243]
  MoveL 2431 to (59.58, 28.56, -3.75) mm, rotated rx 180 ry 0 rz 90 deg; joints [75.256, -16.662, 80.786, 0, 25.876, 75.256]
  MoveC 2432 to (58.62, 31.36, -3.75) mm, rotated rx -180 ry 0 rz 90 deg; joints [75.336, -16.698, 80.912, 0, 25.786, 75.336] to (56.47, 33.39, -3.75) mm, rotated rx 180 ry 0 rz 90 deg; joints [75.383, -16.754, 81.111, 0, 25.643, 75.383]
  MoveC 2433 to (55.64, 33.72, -3.75) mm, rotated rx -180 ry 0 rz 90 deg; joints [75.386, -16.773, 81.179, 0, 25.594, 75.386] to (54.75, 33.82, -3.75) mm, rotated rx 180 ry 0 rz 90 deg; joints [75.382, -16.792, 81.248, 0, 25.545, 75.382]
  MoveL 2434 to (31.18, 33.19, -3.75) mm, rotated rx -180 ry 0 rz 90 deg; joints [75.164, -17.264, 82.963, 0, 24.3, 75.164]
  MoveL 2435 to (31.38, 25.64, -3.75) mm, rotated rx 180 ry 0 rz 90 deg; joints [74.924, -17.22, 82.803, 0, 24.418, 74.924]
  MoveL 2436 to (31.38, 25.64, -0.75) mm, rotated rx 180 ry 0 rz 90 deg; joints [74.924, -17.373, 82.904, 0, 24.469, 74.924]
  Establecer velocidad (1000.0 mm/s)
  MoveL 2437 to (31.38, 25.64, 10) mm, rotated rx -180 ry 0 rz 90 deg; joints [74.924, -17.918, 83.262, 0, 24.656, 74.924]
  Establecer velocidad (66.7 mm/s)
  MoveL 2438 to (67.84, -30.83, 10) mm, rotated rx -180 ry 0 rz 90 deg; joints [73.47, -16.815, 79.386, 0, 27.429, 73.47]
  MoveL 2439 to (67.84, -30.83, -0.5) mm, rotated rx 180 ry 0 rz 90 deg; joints [73.47, -16.29, 79.033, 0, 27.256, 73.47]
  MoveL 2440 to (69.35, -31.02, -0.91) mm, rotated rx -180 ry 0 rz 90 deg; joints [73.478, -16.235, 78.902, 0, 27.333, 73.478]
  MoveL 2441 to (70.86, -30.83, -1.31) mm, rotated rx -180 ry 0 rz 90 deg; joints [73.498, -16.182, 78.778, 0, 27.404, 73.498]
  MoveL 2442 to (72.29, -30.32, -1.72) mm, rotated rx -180 ry 0 rz 90 deg; joints [73.526, -16.133, 78.668, 0, 27.465, 73.526]
  MoveL 2443 to (73.57, -29.5, -2.13) mm, rotated rx 180 ry 0 rz 90 deg; joints [73.563, -16.09, 78.575, 0, 27.514, 73.563]
  MoveL 2444 to (74.64, -28.43, -2.53) mm, rotated rx 180 ry 0 rz 90 deg; joints [73.606, -16.053, 78.505, 0, 27.548, 73.606]
  MoveL 2445 to (75.44, -27.13, -2.94) mm, rotated rx -180 ry 0 rz 90 deg; joints [73.653, -16.023, 78.459, 0, 27.564, 73.653]
  MoveL 2446 to (75.94, -25.7, -3.34) mm, rotated rx 180 ry 0 rz 90 deg; joints [73.702, -16.001, 78.439, 0, 27.562, 73.702]
  MoveL 2447 to (76.08, -24.19, -3.75) mm, rotated rx 180 ry 0 rz 90 deg; joints [73.75, -15.987, 78.448, 0, 27.539, 73.75]
  MoveL 2448 to (76.08, -4.26, -3.75) mm, rotated rx 180 ry 0 rz 90 deg; joints [74.367, -16.114, 78.88, 0, 27.234, 74.367]
  MoveL 2449 to (76.05, -3.82, -3.75) mm, rotated rx -180 ry 0 rz 90 deg; joints [74.381, -16.117, 78.891, 0, 27.227, 74.381]
  MoveC 2450 to (73.49, -0.69, -3.75) mm, rotated rx -180 ry 0 rz 90 deg; joints [74.456, -16.193, 79.151, 0, 27.043, 74.456] to (69.65, 0.6, -3.75) mm, rotated rx -180 ry 0 rz 90 deg; joints [74.463, -16.285, 79.467, 0, 26.818, 74.463]
  MoveC 2451 to (68.44, 0.46, -3.75) mm, rotated rx 180 ry 0 rz 90 deg; joints [74.448, -16.311, 79.555, 0, 26.755, 74.448] to (67.31, -0.02, -3.75) mm, rotated rx -180 ry 0 rz 90 deg; joints [74.423, -16.332, 79.63, 0, 26.702, 74.423]
  MoveL 2452 to (66.25, -1.42, -3.75) mm, rotated rx -180 ry 0 rz 90 deg; joints [74.37, -16.347, 79.68, 0, 26.667, 74.37]
  MoveL 2453 to (53.54, -18.86, -3.75) mm, rotated rx -180 ry 0 rz 90 deg; joints [73.711, -16.512, 80.256, 0, 26.256, 73.711]
  MoveL 2454 to (50.38, -23.22, -3.75) mm, rotated rx 180 ry 0 rz 90 deg; joints [73.546, -16.552, 80.396, 0, 26.156, 73.546]
  MoveC 2455 to (49.53, -26.3, -3.75) mm, rotated rx 180 ry 0 rz 90 deg; joints [73.442, -16.55, 80.391, 0, 26.159, 73.442] to (50.7, -29.28, -3.75) mm, rotated rx 180 ry 0 rz 90 deg; joints [73.36, -16.507, 80.239, 0, 26.268, 73.36]
  MoveL 2456 to (51.65, -30.38, -3.75) mm, rotated rx -180 ry 0 rz 90 deg; joints [73.334, -16.48, 80.144, 0, 26.336, 73.334]
  MoveL 2457 to (67.41, -48.19, -3.75) mm, rotated rx 180 ry 0 rz 90 deg; joints [72.93, -16.02, 78.561, 0, 27.46, 72.93]
  MoveC 2458 to (68.04, -48.69, -3.75) mm, rotated rx 180 ry 0 rz 90 deg; joints [72.921, -16.003, 78.501, 0, 27.502, 72.921] to (68.81, -48.94, -3.75) mm, rotated rx -180 ry 0 rz 90 deg; joints [72.921, -15.984, 78.438, 0, 27.546, 72.921]
  MoveL 2459 to (69.65, -49.06, -3.75) mm, rotated rx -180 ry 0 rz 90 deg; joints [72.925, -15.964, 78.371, 0, 27.593, 72.925]
  MoveL 2460 to (70, -49.04, -3.75) mm, rotated rx -180 ry 0 rz 90 deg; joints [72.929, -15.957, 78.345, 0, 27.612, 72.929]
  MoveC 2461 to (73.7, -47.71, -3.75) mm, rotated rx 180 ry 0 rz 90 deg; joints [73.004, -15.883, 78.096, 0, 27.787, 73.004] to (76.05, -44.56, -3.75) mm, rotated rx 180 ry 0 rz 90 deg; joints [73.123, -15.852, 77.99, 0, 27.861, 73.123]
  MoveL 2462 to (76.08, -43.55, -3.75) mm, rotated rx 180 ry 0 rz 90 deg; joints [73.154, -15.858, 78.011, 0, 27.847, 73.154]
  MoveL 2463 to (76.08, -24.19, -3.75) mm, rotated rx 180 ry 0 rz 90 deg; joints [73.75, -15.987, 78.448, 0, 27.539, 73.75]
  MoveL 2464 to (68.53, -24.19, -3.75) mm, rotated rx -180 ry 0 rz 90 deg; joints [73.682, -16.155, 79.019, 0, 27.136, 73.682]
  MoveL 2465 to (68.53, -24.19, -0.75) mm, rotated rx 180 ry 0 rz 90 deg; joints [73.682, -16.305, 79.121, 0, 27.184, 73.682]
  Establecer velocidad (1000.0 mm/s)
  MoveL 2466 to (68.53, -24.19, 10) mm, rotated rx 180 ry 0 rz 90 deg; joints [73.682, -16.843, 79.482, 0, 27.362, 73.682]
  Establecer velocidad (66.7 mm/s)
  MoveL 2467 to (18.99, -69.39, 10) mm, rotated rx 180 ry 0 rz 90 deg; joints [71.796, -17.596, 82.101, 0, 25.496, 71.796]
  MoveL 2468 to (18.99, -69.39, -0.5) mm, rotated rx -180 ry 0 rz 90 deg; joints [71.796, -17.066, 81.75, 0, 25.316, 71.796]
  MoveL 2469 to (18.83, -70.89, -0.91) mm, rotated rx 180 ry 0 rz 90 deg; joints [71.747, -17.039, 81.712, 0, 25.326, 71.747]
  MoveL 2470 to (19.02, -72.4, -1.31) mm, rotated rx -180 ry 0 rz 90 deg; joints [71.702, -17.004, 81.648, 0, 25.356, 71.702]
  MoveL 2471 to (19.55, -73.82, -1.72) mm, rotated rx 180 ry 0 rz 90 deg; joints [71.663, -16.963, 81.562, 0, 25.401, 71.663]
  MoveL 2472 to (20.38, -75.1, -2.13) mm, rotated rx -180 ry 0 rz 90 deg; joints [71.632, -16.918, 81.458, 0, 25.46, 71.632]
  MoveL 2473 to (21.47, -76.15, -2.53) mm, rotated rx -180 ry 0 rz 90 deg; joints [71.61, -16.868, 81.34, 0, 25.528, 71.61]
  MoveL 2474 to (22.77, -76.95, -2.94) mm, rotated rx -180 ry 0 rz 90 deg; joints [71.599, -16.816, 81.213, 0, 25.603, 71.599]
  MoveL 2475 to (24.21, -77.43, -3.34) mm, rotated rx -180 ry 0 rz 90 deg; joints [71.599, -16.762, 81.082, 0, 25.68, 71.599]
  MoveL 2476 to (25.72, -77.55, -3.75) mm, rotated rx 180 ry 0 rz 90 deg; joints [71.61, -16.71, 80.955, 0, 25.755, 71.61]
  MoveL 2477 to (53.54, -77.26, -3.75) mm, rotated rx -180 ry 0 rz 90 deg; joints [71.903, -16.123, 78.91, 0, 27.213, 71.903]
  MoveL 2478 to (54.18, -77.21, -3.75) mm, rotated rx -180 ry 0 rz 90 deg; joints [71.91, -16.109, 78.864, 0, 27.246, 71.91]
  MoveC 2479 to (55.35, -76.94, -3.75) mm, rotated rx -180 ry 0 rz 90 deg; joints [71.93, -16.086, 78.782, 0, 27.303, 71.93] to (56.38, -76.31, -3.75) mm, rotated rx -180 ry 0 rz 90 deg; joints [71.96, -16.067, 78.721, 0, 27.347, 71.96]
  MoveC 2480 to (58.37, -73.28, -3.75) mm, rotated rx 180 ry 0 rz 90 deg; joints [72.073, -16.045, 78.645, 0, 27.4, 72.073] to (58.43, -69.65, -3.75) mm, rotated rx -180 ry 0 rz 90 deg; joints [72.184, -16.07, 78.729, 0, 27.341, 72.184]
  MoveC 2481 to (58, -68.87, -3.75) mm, rotated rx 180 ry 0 rz 90 deg; joints [72.204, -16.085, 78.78, 0, 27.305, 72.204] to (57.47, -68.15, -3.75) mm, rotated rx -180 ry 0 rz 90 deg; joints [72.221, -16.101, 78.837, 0, 27.264, 72.221]
  MoveL 2482 to (28.9, -35.09, -3.75) mm, rotated rx 180 ry 0 rz 90 deg; joints [72.971, -16.921, 81.712, 0, 25.21, 72.971]
  MoveL 2483 to (27.75, -33.8, -3.75) mm, rotated rx 180 ry 0 rz 90 deg; joints [73, -16.953, 81.824, 0, 25.128, 73]
  MoveL 2484 to (12.79, -21.85, -3.75) mm, rotated rx 180 ry 0 rz 90 deg; joints [73.235, -17.318, 83.166, 0, 24.152, 73.235]
  MoveC 2485 to (11.36, -20.96, -3.75) mm, rotated rx -180 ry 0 rz 90 deg; joints [73.25, -17.351, 83.288, 0, 24.063, 73.25] to (9.77, -20.39, -3.75) mm, rotated rx 180 ry 0 rz 90 deg; joints [73.253, -17.385, 83.414, 0, 23.97, 73.253]
  MoveC 2486 to (5.94, -20.91, -3.75) mm, rotated rx 180 ry 0 rz 90 deg; joints [73.199, -17.455, 83.677, 0, 23.778, 73.199] to (3.51, -23.9, -3.75) mm, rotated rx 180 ry 0 rz 90 deg; joints [73.08, -17.483, 83.785, 0, 23.699, 73.08]
  MoveL 2487 to (3.14, -25.11, -3.75) mm, rotated rx 180 ry 0 rz 90 deg; joints [73.037, -17.484, 83.785, 0, 23.698, 73.037]
  MoveL 2488 to (-8.82, -70.13, -3.75) mm, rotated rx 180 ry 0 rz 90 deg; joints [71.482, -17.437, 83.612, 0, 23.826, 71.482]
  MoveC 2489 to (-9.04, -71.3, -3.75) mm, rotated rx -180 ry 0 rz 90 deg; joints [71.442, -17.434, 83.6, 0, 23.834, 71.442] to (-9.11, -72.48, -3.75) mm, rotated rx 180 ry 0 rz 90 deg; joints [71.404, -17.428, 83.577, 0, 23.851, 71.404]
  MoveC 2490 to (-8.3, -75.21, -3.75) mm, rotated rx 180 ry 0 rz 90 deg; joints [71.327, -17.396, 83.455, 0, 23.941, 71.327] to (-6.17, -77.09, -3.75) mm, rotated rx -180 ry 0 rz 90 deg; joints [71.29, -17.343, 83.259, 0, 24.084, 71.29]
  MoveC 2491 to (-4.5, -77.67, -3.75) mm, rotated rx 180 ry 0 rz 90 deg; joints [71.289, -17.308, 83.126, 0, 24.182, 71.289] to (-2.73, -77.86, -3.75) mm, rotated rx 180 ry 0 rz 90 deg; joints [71.302, -17.273, 82.996, 0, 24.277, 71.302]
  MoveL 2492 to (25.72, -77.55, -3.75) mm, rotated rx 180 ry 0 rz 90 deg; joints [71.61, -16.71, 80.955, 0, 25.755, 71.61]
  MoveL 2493 to (25.64, -70, -3.75) mm, rotated rx 180 ry 0 rz 90 deg; joints [71.845, -16.763, 81.143, 0, 25.62, 71.845]
  MoveL 2494 to (25.64, -70, -0.75) mm, rotated rx 180 ry 0 rz 90 deg; joints [71.845, -16.914, 81.244, 0, 25.67, 71.845]
  Establecer velocidad (1000.0 mm/s)
  MoveL 2495 to (25.64, -70, 10) mm, rotated rx -180 ry 0 rz 90 deg; joints [71.845, -17.456, 81.604, 0, 25.853, 71.845]
  Establecer velocidad (66.7 mm/s)
  MoveL 2496 to (-70.31, -45.34, 10) mm, rotated rx -180 ry 0 rz 90 deg; joints [71.62, -19.355, 88.877, 0, 20.478, 71.62]
  MoveL 2497 to (-70.31, -45.34, -0.5) mm, rotated rx -180 ry 0 rz 90 deg; joints [71.62, -18.809, 88.527, 0, 20.282, 71.62]
  MoveL 2498 to (-71.82, -45.15, -0.91) mm, rotated rx 180 ry 0 rz 90 deg; joints [71.61, -18.813, 88.619, 0, 20.194, 71.61]
  MoveL 2499 to (-73.33, -45.33, -1.31) mm, rotated rx 180 ry 0 rz 90 deg; joints [71.587, -18.814, 88.702, 0, 20.112, 71.587]
  MoveL 2500 to (-74.76, -45.84, -1.72) mm, rotated rx 180 ry 0 rz 90 deg; joints [71.554, -18.813, 88.773, 0, 20.039, 71.554]
  MoveL 2501 to (-76.04, -46.66, -2.13) mm, rotated rx -180 ry 0 rz 90 deg; joints [71.513, -18.807, 88.827, 0, 19.98, 71.513]
  MoveL 2502 to (-77.11, -47.74, -2.53) mm, rotated rx -180 ry 0 rz 90 deg; joints [71.466, -18.797, 88.861, 0, 19.936, 71.466]
  MoveL 2503 to (-77.92, -49.03, -2.94) mm, rotated rx -180 ry 0 rz 90 deg; joints [71.414, -18.782, 88.872, 0, 19.909, 71.414]
  MoveL 2504 to (-78.41, -50.46, -3.34) mm, rotated rx 180 ry 0 rz 90 deg; joints [71.361, -18.761, 88.859, 0, 19.901, 71.361]
  MoveL 2505 to (-78.55, -51.98, -3.75) mm, rotated rx -180 ry 0 rz 90 deg; joints [71.31, -18.734, 88.821, 0, 19.913, 71.31]
  MoveL 2506 to (-78.55, -70.6, -3.75) mm, rotated rx -180 ry 0 rz 90 deg; joints [70.696, -18.634, 88.393, 0, 20.242, 70.696]
  MoveL 2507 to (-78.52, -71.55, -3.75) mm, rotated rx 180 ry 0 rz 90 deg; joints [70.666, -18.628, 88.368, 0, 20.261, 70.666]
  MoveC 2508 to (-76.28, -76.1, -3.75) mm, rotated rx 180 ry 0 rz 90 deg; joints [70.543, -18.568, 88.111, 0, 20.457, 70.543] to (-71.55, -77.92, -3.75) mm, rotated rx 180 ry 0 rz 90 deg; joints [70.538, -18.483, 87.75, 0, 20.732, 70.538]
  MoveL 2509 to (-70.6, -77.92, -3.75) mm, rotated rx -180 ry 0 rz 90 deg; joints [70.549, -18.467, 87.687, 0, 20.781, 70.549]
  MoveL 2510 to (-42.17, -77.7, -3.75) mm, rotated rx -180 ry 0 rz 90 deg; joints [70.878, -17.994, 85.758, 0, 22.236, 70.878]
  MoveL 2511 to (-35.34, -77.64, -3.75) mm, rotated rx 180 ry 0 rz 90 deg; joints [70.955, -17.874, 85.288, 0, 22.586, 70.955]
  MoveC 2512 to (-31.01, -76.13, -3.75) mm, rotated rx 180 ry 0 rz 90 deg; joints [71.051, -17.807, 85.024, 0, 22.783, 71.051] to (-28.48, -72.29, -3.75) mm, rotated rx -180 ry 0 rz 90 deg; joints [71.202, -17.785, 84.94, 0, 22.845, 71.202]
  MoveL 2513 to (-15.94, -24.17, -3.75) mm, rotated rx -180 ry 0 rz 90 deg; joints [72.88, -17.84, 85.153, 0, 22.687, 72.88]
  MoveC 2514 to (-15.6, -22.13, -3.75) mm, rotated rx -180 ry 0 rz 90 deg; joints [72.949, -17.845, 85.173, 0, 22.672, 72.949] to (-15.66, -20.07, -3.75) mm, rotated rx 180 ry 0 rz 90 deg; joints [73.015, -17.857, 85.221, 0, 22.636, 73.015]
  MoveC 2515 to (-17.4, -16.56, -3.75) mm, rotated rx -180 ry 0 rz 90 deg; joints [73.112, -17.907, 85.418, 0, 22.489, 73.112] to (-20.97, -14.91, -3.75) mm, rotated rx 180 ry 0 rz 90 deg; joints [73.13, -17.979, 85.702, 0, 22.278, 73.13]
  MoveC 2516 to (-22.57, -14.89, -3.75) mm, rotated rx 180 ry 0 rz 90 deg; joints [73.115, -18.008, 85.814, 0, 22.193, 73.115] to (-24.17, -15.13, -3.75) mm, rotated rx -180 ry 0 rz 90 deg; joints [73.091, -18.034, 85.92, 0, 22.114, 73.091]
  MoveL 2517 to (-72.49, -25.41, -3.75) mm, rotated rx 180 ry 0 rz 90 deg; joints [72.257, -18.775, 89, 0, 19.775, 72.257]
  MoveL 2518 to (-73.22, -25.59, -3.75) mm, rotated rx 180 ry 0 rz 90 deg; joints [72.243, -18.785, 89.045, 0, 19.74, 72.243]
  MoveC 2519 to (-77.06, -28.08, -3.75) mm, rotated rx -180 ry 0 rz 90 deg; joints [72.119, -18.832, 89.249, 0, 19.583, 72.119] to (-78.55, -32.4, -3.75) mm, rotated rx -180 ry 0 rz 90 deg; joints [71.959, -18.833, 89.255, 0, 19.578, 71.959]
  MoveL 2520 to (-78.55, -51.98, -3.75) mm, rotated rx -180 ry 0 rz 90 deg; joints [71.31, -18.734, 88.821, 0, 19.913, 71.31]
  MoveL 2521 to (-71, -51.98, -3.75) mm, rotated rx -180 ry 0 rz 90 deg; joints [71.394, -18.616, 88.315, 0, 20.301, 71.394]
  MoveL 2522 to (-71, -51.98, -0.75) mm, rotated rx 180 ry 0 rz 90 deg; joints [71.394, -18.772, 88.416, 0, 20.356, 71.394]
  Establecer velocidad (1000.0 mm/s)
  MoveL 2523 to (-71, -51.98, 10) mm, rotated rx 180 ry 0 rz 90 deg; joints [71.394, -19.33, 88.774, 0, 20.557, 71.394]
  Establecer velocidad (66.7 mm/s)
  MoveL 2524 to (-70.31, 36.24, 10) mm, rotated rx -180 ry 0 rz 90 deg; joints [74.351, -19.742, 90.552, 0, 19.189, 74.351]
  MoveL 2525 to (-70.31, 36.24, -0.5) mm, rotated rx 180 ry 0 rz 90 deg; joints [74.351, -19.192, 90.203, 0, 18.989, 74.351]
  MoveL 2526 to (-71.82, 36.42, -0.91) mm, rotated rx 180 ry 0 rz 90 deg; joints [74.343, -19.193, 90.293, 0, 18.9, 74.343]
  MoveL 2527 to (-73.33, 36.24, -1.31) mm, rotated rx 180 ry 0 rz 90 deg; joints [74.323, -19.194, 90.377, 0, 18.816, 74.323]
  MoveL 2528 to (-74.76, 35.73, -1.72) mm, rotated rx -180 ry 0 rz 90 deg; joints [74.292, -19.191, 90.449, 0, 18.742, 74.292]
  MoveL 2529 to (-76.04, 34.91, -2.13) mm, rotated rx 180 ry 0 rz 90 deg; joints [74.251, -19.185, 90.506, 0, 18.679, 74.251]
  MoveL 2530 to (-77.11, 33.83, -2.53) mm, rotated rx -180 ry 0 rz 90 deg; joints [74.204, -19.175, 90.543, 0, 18.632, 74.204]
  MoveL 2531 to (-77.92, 32.54, -2.94) mm, rotated rx -180 ry 0 rz 90 deg; joints [74.153, -19.16, 90.559, 0, 18.601, 74.153]
  MoveL 2532 to (-78.41, 31.1, -3.34) mm, rotated rx 180 ry 0 rz 90 deg; joints [74.099, -19.14, 90.551, 0, 18.589, 74.099]
  MoveL 2533 to (-78.55, 29.6, -3.75) mm, rotated rx 180 ry 0 rz 90 deg; joints [74.046, -19.115, 90.518, 0, 18.596, 74.046]
  MoveL 2534 to (-78.55, 1.42, -3.75) mm, rotated rx 180 ry 0 rz 90 deg; joints [73.092, -18.993, 89.965, 0, 19.028, 73.092]
  MoveL 2535 to (-78.55, 0.47, -3.75) mm, rotated rx 180 ry 0 rz 90 deg; joints [73.06, -18.988, 89.945, 0, 19.043, 73.06]
  MoveC 2536 to (-77.69, -2.87, -3.75) mm, rotated rx -180 ry 0 rz 90 deg; joints [72.956, -18.961, 89.82, 0, 19.141, 72.956] to (-75.34, -5.39, -3.75) mm, rotated rx -180 ry 0 rz 90 deg; joints [72.896, -18.914, 89.611, 0, 19.303, 72.896]
  MoveC 2537 to (-72.56, -6.28, -3.75) mm, rotated rx 180 ry 0 rz 90 deg; joints [72.895, -18.868, 89.407, 0, 19.461, 72.895] to (-69.65, -6.12, -3.75) mm, rotated rx 180 ry 0 rz 90 deg; joints [72.93, -18.824, 89.215, 0, 19.609, 72.93]
  MoveL 2538 to (-20.37, 5.21, -3.75) mm, rotated rx 180 ry 0 rz 90 deg; joints [73.792, -18.074, 86.077, 0, 21.997, 73.792]
  MoveL 2539 to (-19.43, 5.45, -3.75) mm, rotated rx -180 ry 0 rz 90 deg; joints [73.809, -18.058, 86.016, 0, 22.042, 73.809]
  MoveC 2540 to (-15.97, 7.85, -3.75) mm, rotated rx 180 ry 0 rz 90 deg; joints [73.92, -18.01, 85.823, 0, 22.187, 73.92] to (-14.67, 11.85, -3.75) mm, rotated rx -180 ry 0 rz 90 deg; joints [74.063, -18.007, 85.812, 0, 22.195, 74.063]
  MoveC 2541 to (-14.8, 13.29, -3.75) mm, rotated rx 180 ry 0 rz 90 deg; joints [74.109, -18.017, 85.85, 0, 22.167, 74.109] to (-15.17, 14.69, -3.75) mm, rotated rx -180 ry 0 rz 90 deg; joints [74.151, -18.03, 85.904, 0, 22.126, 74.151]
  MoveL 2542 to (-21.89, 33.44, -3.75) mm, rotated rx 180 ry 0 rz 90 deg; joints [74.707, -18.237, 86.737, 0, 21.5, 74.707]
  MoveC 2543 to (-23.06, 35.55, -3.75) mm, rotated rx -180 ry 0 rz 90 deg; joints [74.766, -18.267, 86.858, 0, 21.409, 74.766] to (-24.84, 37.16, -3.75) mm, rotated rx 180 ry 0 rz 90 deg; joints [74.803, -18.305, 87.012, 0, 21.292, 74.803]
  MoveL 2544 to (-65.86, 63.49, -3.75) mm, rotated rx 180 ry 0 rz 90 deg; joints [75.321, -19.065, 90.29, 0, 18.775, 75.321]
  MoveL 2545 to (-67.06, 64.25, -3.75) mm, rotated rx -180 ry 0 rz 90 deg; joints [75.336, -19.085, 90.384, 0, 18.701, 75.336]
  MoveC 2546 to (-69.22, 65.33, -3.75) mm, rotated rx -180 ry 0 rz 90 deg; joints [75.354, -19.121, 90.548, 0, 18.573, 75.354] to (-71.57, 65.92, -3.75) mm, rotated rx 180 ry 0 rz 90 deg; joints [75.353, -19.157, 90.715, 0, 18.442, 75.353]
  MoveC 2547 to (-75.45, 65.13, -3.75) mm, rotated rx -180 ry 0 rz 90 deg; joints [75.291, -19.21, 90.96, 0, 18.25, 75.291] to (-77.97, 62.07, -3.75) mm, rotated rx -180 ry 0 rz 90 deg; joints [75.163, -19.234, 91.074, 0, 18.16, 75.163]
  MoveC 2548 to (-78.41, 60.42, -3.75) mm, rotated rx -180 ry 0 rz 90 deg; joints [75.102, -19.234, 91.074, 0, 18.16, 75.102] to (-78.55, 58.72, -3.75) mm, rotated rx 180 ry 0 rz 90 deg; joints [75.042, -19.23, 91.054, 0, 18.176, 75.042]
  MoveL 2549 to (-78.55, 29.6, -3.75) mm, rotated rx 180 ry 0 rz 90 deg; joints [74.046, -19.115, 90.518, 0, 18.596, 74.046]
  MoveL 2550 to (-71.01, 29.6, -3.75) mm, rotated rx -180 ry 0 rz 90 deg; joints [74.119, -19.004, 90.014, 0, 18.99, 74.119]
  MoveL 2551 to (-71.01, 29.6, -0.75) mm, rotated rx -180 ry 0 rz 90 deg; joints [74.119, -19.161, 90.115, 0, 19.046, 74.119]
  Establecer velocidad (1000.0 mm/s)
  MoveL 2552 to (-71.01, 29.6, 10) mm, rotated rx -180 ry 0 rz 90 deg; joints [74.119, -19.724, 90.473, 0, 19.251, 74.119]
  Establecer velocidad (66.7 mm/s)
  MoveL 2553 to (-69.99, 36.24, 10) mm, rotated rx -180 ry 0 rz 90 deg; joints [74.354, -19.737, 90.531, 0, 19.206, 74.354]
  MoveL 2554 to (-69.99, 36.24, -0.75) mm, rotated rx -180 ry 0 rz 90 deg; joints [74.354, -19.174, 90.173, 0, 19.001, 74.354]
  MoveL 2555 to (-71.5, 36.42, -1.16) mm, rotated rx 180 ry 0 rz 90 deg; joints [74.346, -19.175, 90.263, 0, 18.912, 74.346]
  MoveL 2556 to (-73, 36.24, -1.56) mm, rotated rx -180 ry 0 rz 90 deg; joints [74.326, -19.176, 90.347, 0, 18.829, 74.326]
  MoveL 2557 to (-74.44, 35.73, -1.97) mm, rotated rx 180 ry 0 rz 90 deg; joints [74.295, -19.173, 90.419, 0, 18.754, 74.295]
  MoveL 2558 to (-75.72, 34.91, -2.37) mm, rotated rx 180 ry 0 rz 90 deg; joints [74.255, -19.167, 90.476, 0, 18.691, 74.255]
  MoveL 2559 to (-76.79, 33.83, -2.78) mm, rotated rx 180 ry 0 rz 90 deg; joints [74.208, -19.157, 90.513, 0, 18.644, 74.208]
  MoveL 2560 to (-77.59, 32.54, -3.19) mm, rotated rx -180 ry 0 rz 90 deg; joints [74.156, -19.142, 90.529, 0, 18.613, 74.156]
  MoveL 2561 to (-78.09, 31.1, -3.59) mm, rotated rx 180 ry 0 rz 90 deg; joints [74.102, -19.122, 90.521, 0, 18.601, 74.102]
  MoveL 2562 to (-78.23, 29.6, -4) mm, rotated rx -180 ry 0 rz 90 deg; joints [74.049, -19.097, 90.488, 0, 18.608, 74.049]
  MoveL 2563 to (-78.23, 1.42, -4) mm, rotated rx -180 ry 0 rz 90 deg; joints [73.095, -18.975, 89.935, 0, 19.04, 73.095]
  MoveL 2564 to (-78.23, 0.47, -4) mm, rotated rx 180 ry 0 rz 90 deg; joints [73.063, -18.97, 89.915, 0, 19.055, 73.063]
  MoveC 2565 to (-77.48, -2.64, -4) mm, rotated rx 180 ry 0 rz 90 deg; joints [72.966, -18.945, 89.802, 0, 19.144, 72.966] to (-75.34, -5.03, -4) mm, rotated rx 180 ry 0 rz 90 deg; joints [72.908, -18.902, 89.61, 0, 19.292, 72.908]
  MoveC 2566 to (-72.57, -5.97, -4) mm, rotated rx -180 ry 0 rz 90 deg; joints [72.905, -18.856, 89.406, 0, 19.451, 72.905] to (-69.65, -5.81, -4) mm, rotated rx 180 ry 0 rz 90 deg; joints [72.94, -18.812, 89.213, 0, 19.599, 72.94]
  MoveL 2567 to (-19.93, 5.62, -4) mm, rotated rx 180 ry 0 rz 90 deg; joints [73.81, -18.055, 86.046, 0, 22.009, 73.81]
  MoveC 2568 to (-15.76, 8.74, -4) mm, rotated rx -180 ry 0 rz 90 deg; joints [73.951, -17.998, 85.818, 0, 22.18, 73.951] to (-15.27, 13.92, -4) mm, rotated rx -180 ry 0 rz 90 deg; joints [74.125, -18.015, 85.887, 0, 22.128, 74.125]
  MoveL 2569 to (-15.84, 15.64, -4) mm, rotated rx 180 ry 0 rz 90 deg; joints [74.176, -18.034, 85.961, 0, 22.073, 74.176]
  MoveL 2570 to (-21.94, 32.69, -4) mm, rotated rx 180 ry 0 rz 90 deg; joints [74.682, -18.222, 86.718, 0, 21.504, 74.682]
  MoveL 2571 to (-22.3, 33.64, -4) mm, rotated rx 180 ry 0 rz 90 deg; joints [74.71, -18.232, 86.761, 0, 21.471, 74.71]
  MoveC 2572 to (-23.44, 35.53, -4) mm, rotated rx -180 ry 0 rz 90 deg; joints [74.762, -18.26, 86.876, 0, 21.384, 74.762] to (-25.11, 36.97, -4) mm, rotated rx 180 ry 0 rz 90 deg; joints [74.795, -18.295, 87.019, 0, 21.276, 74.795]
  MoveL 2573 to (-67.17, 63.96, -4) mm, rotated rx 180 ry 0 rz 90 deg; joints [75.326, -19.073, 90.378, 0, 18.695, 75.326]
  MoveC 2574 to (-69.28, 65.02, -4) mm, rotated rx -180 ry 0 rz 90 deg; joints [75.343, -19.107, 90.538, 0, 18.57, 75.343] to (-71.57, 65.62, -4) mm, rotated rx 180 ry 0 rz 90 deg; joints [75.343, -19.143, 90.701, 0, 18.442, 75.343]
  MoveC 2575 to (-75.22, 64.91, -4) mm, rotated rx -180 ry 0 rz 90 deg; joints [75.286, -19.193, 90.933, 0, 18.26, 75.286] to (-77.63, 62.07, -4) mm, rotated rx -180 ry 0 rz 90 deg; joints [75.166, -19.216, 91.043, 0, 18.173, 75.166]
  MoveC 2576 to (-78.08, 60.47, -4) mm, rotated rx 180 ry 0 rz 90 deg; joints [75.107, -19.217, 91.045, 0, 18.172, 75.107] to (-78.23, 58.81, -4) mm, rotated rx -180 ry 0 rz 90 deg; joints [75.048, -19.213, 91.026, 0, 18.187, 75.048]
  MoveL 2577 to (-78.23, 29.6, -4) mm, rotated rx -180 ry 0 rz 90 deg; joints [74.049, -19.097, 90.488, 0, 18.608, 74.049]
  MoveL 2578 to (-70.68, 29.6, -4) mm, rotated rx -180 ry 0 rz 90 deg; joints [74.123, -18.986, 89.984, 0, 19.002, 74.123]
  MoveL 2579 to (-70.68, 29.6, -1) mm, rotated rx -180 ry 0 rz 90 deg; joints [74.123, -19.143, 90.085, 0, 19.058, 74.123]
  Establecer velocidad (1000.0 mm/s)
  MoveL 2580 to (-70.68, 29.6, 10) mm, rotated rx -180 ry 0 rz 90 deg; joints [74.123, -19.719, 90.451, 0, 19.268, 74.123]
  Establecer velocidad (66.7 mm/s)
  MoveL 2581 to (-39.98, -27.24, 10) mm, rotated rx 180 ry 0 rz 90 deg; joints [72.536, -18.951, 87.213, 0, 21.738, 72.536]
  MoveL 2582 to (-39.98, -27.24, -0.75) mm, rotated rx -180 ry 0 rz 90 deg; joints [72.536, -18.396, 86.855, 0, 21.541, 72.536]
  MoveL 2583 to (-40.11, -25.74, -1.16) mm, rotated rx 180 ry 0 rz 90 deg; joints [72.584, -18.386, 86.883, 0, 21.502, 72.584]
  MoveL 2584 to (-40.6, -24.3, -1.56) mm, rotated rx -180 ry 0 rz 90 deg; joints [72.626, -18.38, 86.934, 0, 21.446, 72.626]
  MoveL 2585 to (-41.4, -23, -1.97) mm, rotated rx -180 ry 0 rz 90 deg; joints [72.661, -18.38, 87.003, 0, 21.377, 72.661]
  MoveL 2586 to (-42.46, -21.92, -2.37) mm, rotated rx -180 ry 0 rz 90 deg; joints [72.685, -18.382, 87.086, 0, 21.296, 72.685]
  MoveL 2587 to (-43.74, -21.09, -2.78) mm, rotated rx -180 ry 0 rz 90 deg; joints [72.699, -18.387, 87.177, 0, 21.21, 72.699]
  MoveL 2588 to (-45.17, -20.58, -3.19) mm, rotated rx -180 ry 0 rz 90 deg; joints [72.702, -18.392, 87.272, 0, 21.12, 72.702]
  MoveL 2589 to (-46.68, -20.39, -3.59) mm, rotated rx 180 ry 0 rz 90 deg; joints [72.692, -18.397, 87.366, 0, 21.031, 72.692]
  MoveL 2590 to (-48.18, -20.56, -4) mm, rotated rx 180 ry 0 rz 90 deg; joints [72.671, -18.4, 87.451, 0, 20.949, 72.671]
  MoveL 2591 to (-72.49, -25.73, -4) mm, rotated rx 180 ry 0 rz 90 deg; joints [72.246, -18.76, 88.985, 0, 19.775, 72.246]
  MoveC 2592 to (-74.72, -26.51, -4) mm, rotated rx -180 ry 0 rz 90 deg; joints [72.196, -18.791, 89.117, 0, 19.674, 72.196] to (-76.58, -27.96, -4) mm, rotated rx 180 ry 0 rz 90 deg; joints [72.128, -18.812, 89.211, 0, 19.601, 72.128]
  MoveC 2593 to (-77.73, -29.72, -4) mm, rotated rx 180 ry 0 rz 90 deg; joints [72.057, -18.821, 89.249, 0, 19.571, 72.057] to (-78.19, -31.78, -4) mm, rotated rx -180 ry 0 rz 90 deg; joints [71.984, -18.818, 89.236, 0, 19.582, 71.984]
  MoveL 2594 to (-78.23, -32.69, -4) mm, rotated rx -180 ry 0 rz 90 deg; joints [71.953, -18.814, 89.218, 0, 19.595, 71.953]
  MoveL 2595 to (-78.23, -71.08, -4) mm, rotated rx 180 ry 0 rz 90 deg; joints [70.684, -18.613, 88.351, 0, 20.262, 70.684]
  MoveC 2596 to (-77.03, -74.82, -4) mm, rotated rx 180 ry 0 rz 90 deg; joints [70.576, -18.574, 88.183, 0, 20.391, 70.576] to (-73.88, -77.16, -4) mm, rotated rx -180 ry 0 rz 90 deg; joints [70.536, -18.511, 87.916, 0, 20.595, 70.536]
  MoveC 2597 to (-72.44, -77.51, -4) mm, rotated rx 180 ry 0 rz 90 deg; joints [70.541, -18.486, 87.812, 0, 20.674, 70.541] to (-70.97, -77.62, -4) mm, rotated rx -180 ry 0 rz 90 deg; joints [70.554, -18.462, 87.71, 0, 20.752, 70.554]
  MoveL 2598 to (-42.17, -77.38, -4) mm, rotated rx -180 ry 0 rz 90 deg; joints [70.888, -17.983, 85.757, 0, 22.225, 70.888]
  MoveL 2599 to (-35.29, -77.32, -4) mm, rotated rx 180 ry 0 rz 90 deg; joints [70.966, -17.863, 85.284, 0, 22.579, 70.966]
  MoveC 2600 to (-31.27, -75.95, -4) mm, rotated rx -180 ry 0 rz 90 deg; joints [71.054, -17.8, 85.038, 0, 22.761, 71.054] to (-28.86, -72.45, -4) mm, rotated rx 180 ry 0 rz 90 deg; joints [71.192, -17.778, 84.954, 0, 22.824, 71.192]
  MoveL 2601 to (-28.6, -71.55, -4) mm, rotated rx -180 ry 0 rz 90 deg; joints [71.224, -17.779, 84.957, 0, 22.822, 71.224]
  MoveL 2602 to (-16.17, -23.83, -4) mm, rotated rx 180 ry 0 rz 90 deg; joints [72.888, -17.833, 85.168, 0, 22.665, 72.888]
  MoveC 2603 to (-15.88, -21.79, -4) mm, rotated rx -180 ry 0 rz 90 deg; joints [72.957, -17.839, 85.191, 0, 22.648, 72.957] to (-16.04, -19.73, -4) mm, rotated rx -180 ry 0 rz 90 deg; joints [73.022, -17.853, 85.246, 0, 22.607, 73.022]
  MoveC 2604 to (-17.86, -16.56, -4) mm, rotated rx 180 ry 0 rz 90 deg; joints [73.107, -17.903, 85.441, 0, 22.461, 73.107] to (-21.25, -15.19, -4) mm, rotated rx 180 ry 0 rz 90 deg; joints [73.118, -17.97, 85.707, 0, 22.263, 73.118]
  MoveC 2605 to (-22.57, -15.21, -4) mm, rotated rx 180 ry 0 rz 90 deg; joints [73.104, -17.993, 85.799, 0, 22.194, 73.104] to (-23.87, -15.4, -4) mm, rotated rx 180 ry 0 rz 90 deg; joints [73.085, -18.015, 85.885, 0, 22.129, 73.085]
  MoveL 2606 to (-48.18, -20.56, -4) mm, rotated rx 180 ry 0 rz 90 deg; joints [72.671, -18.4, 87.451, 0, 20.949, 72.671]
  MoveL 2607 to (-46.61, -27.95, -4) mm, rotated rx 180 ry 0 rz 90 deg; joints [72.445, -18.336, 87.186, 0, 21.15, 72.445]
  MoveL 2608 to (-46.61, -27.95, -1) mm, rotated rx 180 ry 0 rz 90 deg; joints [72.445, -18.491, 87.286, 0, 21.204, 72.445]
  Establecer velocidad (1000.0 mm/s)
  MoveL 2609 to (-46.61, -27.95, 10) mm, rotated rx -180 ry 0 rz 90 deg; joints [72.445, -19.059, 87.652, 0, 21.407, 72.445]
  Establecer velocidad (66.7 mm/s)
  MoveL 2610 to (19.05, -69.08, 10) mm, rotated rx 180 ry 0 rz 90 deg; joints [71.806, -17.597, 82.104, 0, 25.494, 71.806]
  MoveL 2611 to (19.05, -69.08, -0.75) mm, rotated rx -180 ry 0 rz 90 deg; joints [71.806, -17.054, 81.745, 0, 25.31, 71.806]
  MoveL 2612 to (18.88, -70.59, -1.16) mm, rotated rx -180 ry 0 rz 90 deg; joints [71.757, -17.027, 81.707, 0, 25.32, 71.757]
  MoveL 2613 to (19.08, -72.09, -1.56) mm, rotated rx 180 ry 0 rz 90 deg; joints [71.712, -16.992, 81.643, 0, 25.349, 71.712]
  MoveL 2614 to (19.61, -73.52, -1.97) mm, rotated rx 180 ry 0 rz 90 deg; joints [71.673, -16.952, 81.557, 0, 25.395, 71.673]
  MoveL 2615 to (20.44, -74.79, -2.37) mm, rotated rx 180 ry 0 rz 90 deg; joints [71.642, -16.906, 81.453, 0, 25.453, 71.642]
  MoveL 2616 to (21.53, -75.85, -2.78) mm, rotated rx -180 ry 0 rz 90 deg; joints [71.62, -16.856, 81.334, 0, 25.522, 71.62]
  MoveL 2617 to (22.83, -76.64, -3.19) mm, rotated rx -180 ry 0 rz 90 deg; joints [71.609, -16.804, 81.207, 0, 25.597, 71.609]
  MoveL 2618 to (24.27, -77.12, -3.59) mm, rotated rx 180 ry 0 rz 90 deg; joints [71.609, -16.751, 81.077, 0, 25.674, 71.609]
  MoveL 2619 to (25.78, -77.25, -4) mm, rotated rx 180 ry 0 rz 90 deg; joints [71.62, -16.698, 80.95, 0, 25.748, 71.62]
  MoveL 2620 to (53.16, -76.96, -4) mm, rotated rx -180 ry 0 rz 90 deg; joints [71.908, -16.121, 78.937, 0, 27.183, 71.908]
  MoveL 2621 to (53.92, -76.93, -4) mm, rotated rx 180 ry 0 rz 90 deg; joints [71.917, -16.104, 78.881, 0, 27.223, 71.917]
  MoveC 2622 to (54.7, -76.78, -4) mm, rotated rx 180 ry 0 rz 90 deg; joints [71.929, -16.088, 78.826, 0, 27.262, 71.929] to (55.41, -76.42, -4) mm, rotated rx -180 ry 0 rz 90 deg; joints [71.947, -16.075, 78.782, 0, 27.293, 71.947]
